C05487=1208.103,115.471,-50.349,-178.483,5.857,148.589
C05488=1208.098,115.720,-50.368,-178.480,5.858,148.588
C05489=1208.094,115.969,-50.387,-178.477,5.859,148.588
C05490=1208.089,116.219,-50.407,-178.474,5.860,148.587
C05491=1208.084,116.468,-50.426,-178.472,5.861,148.587
C05492=1208.079,116.717,-50.447,-178.469,5.863,148.586
C05493=1208.074,116.965,-50.466,-178.467,5.864,148.586
C05494=1208.070,117.215,-50.485,-178.465,5.865,148.585
C05495=1208.065,117.464,-50.505,-178.461,5.866,148.585
C05496=1208.060,117.713,-50.524,-178.459,5.867,148.584
C05497=1208.055,117.963,-50.543,-178.456,5.868,148.584
C05498=1208.051,118.212,-50.563,-178.454,5.869,148.583
C05499=1208.046,118.461,-50.582,-178.451,5.871,148.583
C05500=1208.041,118.710,-50.602,-178.449,5.872,148.582
C05501=1208.036,118.960,-50.621,-178.446,5.872,148.582
C05502=1208.031,119.209,-50.640,-178.443,5.874,148.581
C05503=1208.026,119.458,-50.660,-178.441,5.875,148.581
C05504=1208.021,119.707,-50.680,-178.438,5.877,148.580
C05505=1208.017,119.956,-50.699,-178.436,5.877,148.580
C05506=1208.013,120.205,-50.719,-178.433,5.879,148.579
C05507=1208.007,120.454,-50.738,-178.431,5.880,148.579
C05508=1208.002,120.704,-50.758,-178.428,5.881,148.578
C05509=1207.998,120.953,-50.778,-178.425,5.882,148.578
C05510=1207.993,121.202,-50.798,-178.423,5.883,148.577
C05511=1207.988,121.451,-50.817,-178.420,5.885,148.577
C05512=1207.983,121.701,-50.837,-178.418,5.885,148.576
C05513=1207.979,121.950,-50.856,-178.415,5.887,148.576
C05514=1207.974,122.198,-50.876,-178.412,5.888,148.575
C05515=1207.969,122.448,-50.895,-178.410,5.889,148.575
C05516=1207.965,122.698,-50.915,-178.407,5.890,148.574
C05517=1207.959,122.946,-50.934,-178.404,5.892,148.574
C05518=1207.955,123.195,-50.955,-178.402,5.893,148.573
C05519=1207.950,123.445,-50.974,-178.399,5.894,148.573
C05520=1207.945,123.694,-50.994,-178.397,5.895,148.572
C05521=1207.940,123.943,-51.014,-178.394,5.897,148.572
C05522=1207.936,124.192,-51.034,-178.392,5.897,148.571
C05523=1207.931,124.442,-51.053,-178.388,5.899,148.571
C05524=1207.926,124.691,-51.074,-178.386,5.900,148.570
C05525=1207.921,124.940,-51.093,-178.384,5.901,148.570
C05526=1207.916,125.189,-51.113,-178.381,5.902,148.569
C05527=1207.912,125.438,-51.133,-178.379,5.903,148.569
C05528=1207.907,125.688,-51.153,-178.376,5.905,148.568
C05529=1207.902,125.937,-51.172,-178.374,5.906,148.568
C05530=1207.897,126.186,-51.192,-178.370,5.907,148.567
C05531=1207.893,126.435,-51.212,-178.368,5.908,148.567
C05532=1207.888,126.684,-51.232,-178.366,5.910,148.566
C05533=1207.883,126.933,-51.252,-178.363,5.910,148.566
C05534=1207.878,127.182,-51.272,-178.360,5.912,148.565
C05535=1207.874,127.431,-51.292,-178.358,5.913,148.565
C05536=1207.869,127.681,-51.311,-178.355,5.914,148.564
C05537=1207.864,127.930,-51.332,-178.353,5.915,148.564
C05538=1207.859,128.179,-51.351,-178.350,5.917,148.563
C05539=1207.855,128.428,-51.371,-178.348,5.918,148.563
C05540=1207.850,128.677,-51.391,-178.344,5.919,148.562
C05541=1207.846,128.926,-51.412,-178.342,5.920,148.562
C05542=1207.841,129.176,-51.431,-178.339,5.922,148.561
C05543=1207.836,129.425,-51.452,-178.337,5.923,148.561
C05544=1207.830,129.674,-51.471,-178.334,5.924,148.560
C05545=1207.826,129.923,-51.492,-178.332,5.925,148.560
C05546=1207.821,130.172,-51.512,-178.329,5.927,148.559
C05547=1207.817,130.421,-51.532,-178.326,5.927,148.559
C05548=1207.812,130.670,-51.552,-178.324,5.929,148.558
C05549=1207.807,130.920,-51.572,-178.322,5.930,148.558
C05550=1207.802,131.169,-51.592,-178.318,5.932,148.557
C05551=1207.797,131.418,-51.613,-178.316,5.933,148.557
C05552=1207.793,131.667,-51.632,-178.313,5.934,148.556
C05553=1207.788,131.916,-51.653,-178.311,5.935,148.556
C05554=1207.783,132.166,-51.672,-178.308,5.937,148.555
C05555=1207.779,132.415,-51.693,-178.306,5.937,148.555
C05556=1207.774,132.664,-51.714,-178.303,5.939,148.554
C05557=1207.769,132.932,-51.735,-178.300,5.941,148.554
C05558=1207.763,133.201,-51.757,-178.298,5.941,148.553
C05559=1207.759,133.469,-51.778,-178.295,5.943,148.553
C05560=1207.753,133.738,-51.801,-178.292,5.945,148.552
C05561=1207.748,133.987,-51.820,-178.289,5.945,148.552
C05562=1207.744,134.236,-51.841,-178.287,5.947,148.551
C05563=1207.739,134.486,-51.862,-178.285,5.948,148.551
C05564=1207.734,134.735,-51.881,-178.281,5.950,148.550
C05565=1207.730,134.984,-51.902,-178.279,5.951,148.550
C05566=1207.725,135.233,-51.922,-178.276,5.952,148.549
C05567=1207.719,135.482,-51.943,-178.273,5.954,148.549
C05568=1207.715,135.731,-51.962,-178.271,5.955,148.549
C05569=1207.710,135.980,-51.983,-178.268,5.956,148.548
C05570=1207.705,136.229,-52.004,-178.266,5.957,148.548
C05571=1207.701,136.478,-52.024,-178.263,5.959,148.547
C05572=1207.696,136.727,-52.045,-178.261,5.959,148.547
C05573=1207.691,136.977,-52.064,-178.258,5.961,148.546
C05574=1207.686,137.226,-52.085,-178.255,5.962,148.546
C05575=1207.682,137.475,-52.106,-178.253,5.964,148.545
C05576=1207.677,137.724,-52.126,-178.250,5.965,148.545
C05577=1207.672,137.973,-52.147,-178.247,5.966,148.544
C05578=1207.668,138.222,-52.167,-178.245,5.968,148.544
C05579=1207.663,138.471,-52.188,-178.243,5.969,148.543
C05580=1207.658,138.720,-52.209,-178.239,5.970,148.543
C05581=1207.653,138.970,-52.228,-178.237,5.971,148.542
C05582=1207.648,139.219,-52.249,-178.235,5.973,148.542
C05583=1207.644,139.468,-52.270,-178.232,5.974,148.541
C05584=1207.639,139.717,-52.290,-178.229,5.975,148.541
C05585=1207.634,139.966,-52.311,-178.227,5.977,148.541
C05586=1207.630,140.215,-52.331,-178.224,5.978,148.540
C05587=1207.625,140.464,-52.352,-178.221,5.980,148.540
C05588=1207.620,140.714,-52.373,-178.219,5.981,148.539
C05589=1207.616,140.962,-52.393,-178.216,5.982,148.539
C05590=1207.611,141.212,-52.414,-178.214,5.983,148.538
C05591=1207.606,141.461,-52.434,-178.211,5.985,148.538
C05592=1207.601,141.710,-52.455,-178.208,5.986,148.537
C05593=1207.597,141.959,-52.476,-178.206,5.987,148.537
C05594=1207.592,142.208,-52.496,-178.203,5.989,148.536
C05595=1207.587,142.457,-52.517,-178.201,5.990,148.536
C05596=1207.582,142.706,-52.537,-178.198,5.991,148.535
C05597=1207.577,142.955,-52.558,-178.195,5.993,148.535
C05598=1207.573,143.204,-52.579,-178.193,5.994,148.534
C05599=1207.568,143.454,-52.600,-178.190,5.996,148.534
C05600=1207.563,143.702,-52.620,-178.188,5.996,148.534
C05601=1207.559,143.952,-52.642,-178.185,5.998,148.533
C05602=1207.555,144.201,-52.662,-178.182,6.000,148.533
C05603=1207.549,144.450,-52.683,-178.180,6.001,148.532
C05604=1207.545,144.699,-52.704,-178.177,6.002,148.532
C05605=1207.540,144.948,-52.725,-178.175,6.003,148.531
C05606=1207.535,145.197,-52.745,-178.172,6.005,148.531
C05607=1207.530,145.446,-52.766,-178.169,6.006,148.530
C05608=1207.526,145.695,-52.787,-178.167,6.007,148.530
C05609=1207.521,145.944,-52.808,-178.164,6.009,148.529
C05610=1207.516,146.193,-52.829,-178.162,6.010,148.529
C05611=1207.512,146.443,-52.850,-178.159,6.012,148.528
C05612=1207.507,146.692,-52.871,-178.156,6.013,148.528
C05613=1207.503,146.941,-52.892,-178.154,6.014,148.528
C05614=1207.497,147.190,-52.913,-178.151,6.016,148.527
C05615=1207.493,147.439,-52.933,-178.149,6.017,148.527
C05616=1207.488,147.688,-52.954,-178.146,6.018,148.526
C05617=1207.483,147.937,-52.976,-178.143,6.020,148.526
C05618=1207.478,148.186,-52.996,-178.141,6.021,148.525
C05619=1207.474,148.436,-53.018,-178.138,6.023,148.525
C05620=1207.469,148.685,-53.039,-178.136,6.024,148.525
C05621=1207.465,148.933,-53.060,-178.133,6.025,148.524
C05622=1207.459,149.182,-53.081,-178.130,6.027,148.524
C05623=1207.455,149.431,-53.101,-178.128,6.028,148.523
C05624=1207.450,149.680,-53.123,-178.125,6.029,148.523
C05625=1207.446,149.930,-53.144,-178.122,6.031,148.522
C05626=1207.441,150.179,-53.164,-178.120,6.032,148.522
C05627=1207.436,150.428,-53.186,-178.118,6.034,148.521
C05628=1207.431,150.677,-53.207,-178.114,6.035,148.521
C05629=1207.427,150.925,-53.228,-178.112,6.036,148.520
C05630=1207.422,151.175,-53.249,-178.110,6.038,148.520
C05631=1207.417,151.424,-53.270,-178.107,6.039,148.519
C05632=1207.412,151.673,-53.292,-178.104,6.041,148.519
C05633=1207.408,151.922,-53.313,-178.102,6.042,148.519
C05634=1207.403,152.171,-53.334,-178.100,6.043,148.518
C05635=1207.398,152.421,-53.356,-178.096,6.045,148.518
C05636=1207.394,152.669,-53.377,-178.094,6.047,148.517
C05637=1207.389,152.918,-53.398,-178.092,6.047,148.517
C05638=1207.384,153.167,-53.419,-178.089,6.049,148.517
C05639=1207.380,153.417,-53.441,-178.086,6.051,148.516
C05640=1207.374,153.666,-53.462,-178.084,6.052,148.516
C05641=1207.370,153.914,-53.483,-178.081,6.054,148.515
C05642=1207.365,154.163,-53.504,-178.078,6.055,148.515
C05643=1207.361,154.413,-53.526,-178.076,6.056,148.514
C05644=1207.356,154.662,-53.547,-178.073,6.058,148.514
C05645=1207.351,154.911,-53.568,-178.070,6.060,148.513
C05646=1207.347,155.159,-53.589,-178.068,6.061,148.513
C05647=1207.342,155.409,-53.611,-178.065,6.062,148.512
C05648=1207.337,155.658,-53.632,-178.063,6.064,148.512
C05649=1207.332,155.907,-53.653,-178.060,6.065,148.512
C05650=1207.327,156.156,-53.675,-178.058,6.067,148.511
C05651=1207.323,156.405,-53.697,-178.055,6.068,148.511
C05652=1207.319,156.654,-53.717,-178.052,6.069,148.510
C05653=1207.314,156.903,-53.739,-178.050,6.071,148.510
C05654=1207.309,157.153,-53.760,-178.047,6.073,148.510
C05655=1207.304,157.401,-53.782,-178.045,6.073,148.509
C05656=1207.299,157.650,-53.804,-178.042,6.075,148.509
C05657=1207.295,157.900,-53.825,-178.039,6.077,148.508
C05658=1207.290,158.148,-53.847,-178.037,6.078,148.508
C05659=1207.285,158.397,-53.869,-178.034,6.079,148.507
C05660=1207.282,158.646,-53.890,-178.031,6.081,148.507
C05661=1207.276,158.915,-53.913,-178.029,6.083,148.506
C05662=1207.270,159.184,-53.936,-178.025,6.084,148.506
C05663=1207.265,159.453,-53.959,-178.023,6.086,148.505
C05664=1207.260,159.722,-53.983,-178.021,6.087,148.505
C05665=1207.256,159.971,-54.005,-178.018,6.089,148.505
C05666=1207.251,160.221,-54.026,-178.015,6.090,148.504
C05667=1207.247,160.470,-54.048,-178.012,6.092,148.504
C05668=1207.242,160.718,-54.069,-178.010,6.093,148.503
C05669=1207.237,160.967,-54.091,-178.007,6.095,148.503
C05670=1207.233,161.217,-54.112,-178.004,6.096,148.502
C05671=1207.228,161.465,-54.134,-178.002,6.097,148.502
C05672=1207.223,161.714,-54.156,-177.999,6.099,148.502
C05673=1207.219,161.963,-54.178,-177.997,6.101,148.501
C05674=1207.214,162.212,-54.199,-177.994,6.102,148.501
C05675=1207.210,162.461,-54.222,-177.992,6.103,148.500
C05676=1207.205,162.710,-54.243,-177.989,6.105,148.500
C05677=1207.200,162.959,-54.264,-177.986,6.107,148.500
C05678=1207.195,163.209,-54.286,-177.984,6.108,148.499
C05679=1207.190,163.457,-54.308,-177.981,6.109,148.499
C05680=1207.185,163.707,-54.331,-177.978,6.111,148.498
C05681=1207.181,163.956,-54.352,-177.976,6.113,148.498
C05682=1207.176,164.205,-54.374,-177.974,6.114,148.497
C05683=1207.171,164.454,-54.396,-177.971,6.116,148.497
C05684=1207.167,164.702,-54.418,-177.968,6.117,148.496
C05685=1207.162,164.952,-54.440,-177.966,6.118,148.496
C05686=1207.157,165.200,-54.461,-177.963,6.120,148.496
C05687=1207.153,165.450,-54.483,-177.960,6.122,148.495
C05688=1207.148,165.698,-54.505,-177.958,6.124,148.495
C05689=1207.144,165.947,-54.527,-177.955,6.124,148.494
C05690=1207.139,166.196,-54.549,-177.952,6.126,148.494
C05691=1207.135,166.445,-54.571,-177.950,6.128,148.494
C05692=1207.129,166.694,-54.593,-177.947,6.130,148.493
C05693=1207.125,166.944,-54.615,-177.945,6.131,148.493
C05694=1207.120,167.192,-54.637,-177.942,6.132,148.493
C05695=1207.116,167.442,-54.659,-177.939,6.134,148.492
C05696=1207.111,167.690,-54.681,-177.936,6.136,148.492
C05697=1207.107,167.940,-54.703,-177.934,6.137,148.491
C05698=1207.101,168.189,-54.725,-177.932,6.139,148.491
C05699=1207.097,168.438,-54.747,-177.929,6.140,148.490
C05700=1207.092,168.686,-54.769,-177.926,6.142,148.490
C05701=1207.088,168.935,-54.791,-177.924,6.143,148.489
C05702=1207.083,169.184,-54.813,-177.921,6.145,148.489
C05703=1207.078,169.434,-54.836,-177.918,6.146,148.489
C05704=1207.073,169.682,-54.857,-177.916,6.148,148.488
C05705=1207.069,169.932,-54.879,-177.914,6.149,148.488
C05706=1207.064,170.180,-54.901,-177.911,6.151,148.488
C05707=1207.060,170.429,-54.924,-177.908,6.152,148.487
C05708=1207.055,170.678,-54.946,-177.905,6.154,148.487
C05709=1207.050,170.927,-54.968,-177.903,6.155,148.486
C05710=1207.045,171.176,-54.990,-177.900,6.157,148.486
C05711=1207.041,171.425,-55.013,-177.898,6.159,148.486
C05712=1207.036,171.674,-55.035,-177.895,6.161,148.485
C05713=1207.032,171.923,-55.057,-177.892,6.162,148.485
C05714=1207.027,172.172,-55.079,-177.890,6.163,148.484
C05715=1207.022,172.421,-55.102,-177.887,6.165,148.484
C05716=1207.018,172.670,-55.124,-177.884,6.167,148.484
C05717=1207.013,172.919,-55.146,-177.882,6.169,148.483
C05718=1207.008,173.168,-55.168,-177.880,6.170,148.483
C05719=1207.003,173.416,-55.191,-177.877,6.171,148.482
C05720=1206.999,173.666,-55.213,-177.874,6.173,148.482
C05721=1206.994,173.915,-55.236,-177.871,6.175,148.481
C05722=1206.989,174.163,-55.258,-177.869,6.176,148.481
C05723=1206.985,174.413,-55.280,-177.866,6.177,148.481
C05724=1206.980,174.662,-55.303,-177.864,6.179,148.480
C05725=1206.976,174.910,-55.325,-177.861,6.181,148.480
C05726=1206.971,175.160,-55.347,-177.859,6.183,148.480
C05727=1206.966,175.408,-55.370,-177.856,6.185,148.479
C05728=1206.962,175.657,-55.392,-177.854,6.186,148.479
C05729=1206.957,175.907,-55.415,-177.851,6.187,148.478
C05730=1206.952,176.155,-55.437,-177.848,6.189,148.478
C05731=1206.948,176.404,-55.459,-177.845,6.191,148.478
C05732=1206.943,176.653,-55.483,-177.843,6.193,148.477
C05733=1206.938,176.902,-55.504,-177.841,6.193,148.477
C05734=1206.934,177.151,-55.528,-177.838,6.195,148.476
C05735=1206.929,177.400,-55.550,-177.835,6.197,148.476
C05736=1206.925,177.648,-55.572,-177.833,6.199,148.476
C05737=1206.920,177.898,-55.595,-177.830,6.201,148.475
C05738=1206.916,178.147,-55.617,-177.827,6.201,148.475
C05739=1206.910,178.396,-55.640,-177.825,6.203,148.474
C05740=1206.906,178.644,-55.662,-177.822,6.205,148.474
C05741=1206.901,178.894,-55.685,-177.819,6.207,148.474
C05742=1206.897,179.142,-55.708,-177.817,6.209,148.473
C05743=1206.892,179.391,-55.731,-177.814,6.210,148.473
C05744=1206.888,179.640,-55.753,-177.812,6.211,148.473
C05745=1206.882,179.889,-55.776,-177.809,6.213,148.472
C05746=1206.878,180.138,-55.798,-177.807,6.215,148.472
C05747=1206.874,180.387,-55.821,-177.804,6.217,148.472
C05748=1206.870,180.636,-55.844,-177.801,6.219,148.471
C05749=1206.864,180.885,-55.866,-177.798,6.220,148.471
C05750=1206.860,181.134,-55.889,-177.796,6.221,148.470
C05751=1206.855,181.383,-55.912,-177.793,6.223,148.470
C05752=1206.851,181.632,-55.935,-177.791,6.225,148.470
C05753=1206.846,181.880,-55.958,-177.788,6.227,148.469
C05754=1206.841,182.129,-55.981,-177.785,6.228,148.469
C05755=1206.837,182.379,-56.003,-177.783,6.230,148.468
C05756=1206.832,182.628,-56.026,-177.781,6.231,148.468
C05757=1206.827,182.876,-56.049,-177.778,6.233,148.468
C05758=1206.822,183.125,-56.071,-177.775,6.235,148.467
C05759=1206.818,183.374,-56.095,-177.773,6.237,148.467
C05760=1206.814,183.623,-56.117,-177.770,6.238,148.467
C05761=1206.809,183.871,-56.140,-177.767,6.240,148.466
C05762=1206.804,184.121,-56.163,-177.764,6.242,148.466
C05763=1206.800,184.370,-56.186,-177.762,6.243,148.465
C05764=1206.795,184.619,-56.209,-177.759,6.245,148.465
C05765=1206.790,184.888,-56.234,-177.757,6.246,148.465
C05766=1206.785,185.158,-56.259,-177.754,6.248,148.464
C05767=1206.780,185.428,-56.284,-177.751,6.251,148.464
C05768=1206.775,185.697,-56.308,-177.748,6.252,148.463
C05769=1206.770,185.946,-56.332,-177.745,6.254,148.463
C05770=1206.766,186.195,-56.355,-177.743,6.255,148.463
C05771=1206.761,186.443,-56.377,-177.740,6.257,148.462
C05772=1206.756,186.692,-56.401,-177.738,6.259,148.462
C05773=1206.752,186.941,-56.424,-177.735,6.261,148.462
C05774=1206.748,187.190,-56.447,-177.732,6.262,148.461
C05775=1206.743,187.439,-56.470,-177.730,6.264,148.461
C05776=1206.738,187.689,-56.493,-177.727,6.266,148.461
C05777=1206.733,187.937,-56.516,-177.724,6.268,148.460
C05778=1206.729,188.186,-56.539,-177.722,6.269,148.460
C05779=1206.724,188.435,-56.562,-177.720,6.271,148.459
C05780=1206.719,188.684,-56.585,-177.717,6.272,148.459
C05781=1206.715,188.933,-56.609,-177.714,6.274,148.459
C05782=1206.711,189.182,-56.631,-177.712,6.276,148.458
C05783=1206.706,189.431,-56.655,-177.709,6.278,148.458
C05784=1206.701,189.680,-56.678,-177.706,6.280,148.458
C05785=1206.696,189.928,-56.701,-177.704,6.282,148.457
C05786=1206.691,190.177,-56.724,-177.701,6.283,148.457
C05787=1206.687,190.426,-56.747,-177.699,6.284,148.457
C05788=1206.683,190.675,-56.771,-177.696,6.286,148.456
C05789=1206.678,190.924,-56.794,-177.694,6.288,148.456
C05790=1206.674,191.172,-56.818,-177.691,6.290,148.456
C05791=1206.669,191.421,-56.841,-177.688,6.292,148.455
C05792=1206.664,191.670,-56.865,-177.686,6.293,148.455
C05793=1206.660,191.919,-56.887,-177.683,6.295,148.455
C05794=1206.655,192.168,-56.911,-177.680,6.297,148.454
C05795=1206.651,192.417,-56.934,-177.678,6.299,148.454
C05796=1206.645,192.666,-56.957,-177.675,6.301,148.454
C05797=1206.641,192.915,-56.981,-177.672,6.303,148.453
C05798=1206.636,193.163,-57.005,-177.670,6.304,148.453
C05799=1206.632,193.412,-57.028,-177.668,6.305,148.452
C05800=1206.627,193.661,-57.051,-177.665,6.307,148.452
C05801=1206.622,193.910,-57.075,-177.662,6.309,148.452
C05802=1206.618,194.159,-57.097,-177.660,6.311,148.451
C05803=1206.614,194.408,-57.121,-177.657,6.313,148.451
C05804=1206.609,194.656,-57.145,-177.654,6.314,148.451
C05805=1206.605,194.905,-57.168,-177.652,6.316,148.450
C05806=1206.600,195.154,-57.192,-177.649,6.318,148.450
C05807=1206.595,195.403,-57.215,-177.647,6.320,148.450
C05808=1206.591,195.652,-57.239,-177.644,6.322,148.449
C05809=1206.586,195.901,-57.262,-177.641,6.324,148.449
C05810=1206.581,196.150,-57.286,-177.639,6.325,148.449
C05811=1206.577,196.398,-57.310,-177.636,6.326,148.448
C05812=1206.572,196.647,-57.333,-177.634,6.328,148.448
C05813=1206.568,196.896,-57.357,-177.631,6.330,148.448
C05814=1206.563,197.145,-57.381,-177.629,6.332,148.447
C05815=1206.558,197.394,-57.404,-177.626,6.334,148.447
C05816=1206.554,197.643,-57.427,-177.623,6.336,148.447
C05817=1206.549,197.891,-57.451,-177.621,6.337,148.446
C05818=1206.545,198.140,-57.475,-177.618,6.339,148.446
C05819=1206.540,198.389,-57.498,-177.615,6.341,148.445
C05820=1206.536,198.638,-57.522,-177.613,6.343,148.445
C05821=1206.531,198.887,-57.546,-177.610,6.345,148.445
C05822=1206.526,199.135,-57.570,-177.607,6.346,148.444
C05823=1206.522,199.385,-57.594,-177.605,6.348,148.444
C05824=1206.517,199.634,-57.618,-177.602,6.350,148.444
C05825=1206.513,199.883,-57.641,-177.599,6.352,148.443
C05826=1206.508,200.131,-57.665,-177.597,6.354,148.443
C05827=1206.503,200.380,-57.689,-177.594,6.356,148.443
C05828=1206.499,200.629,-57.712,-177.591,6.357,148.442
C05829=1206.494,200.877,-57.736,-177.589,6.359,148.442
C05830=1206.490,201.126,-57.760,-177.586,6.361,148.442
C05831=1206.485,201.375,-57.784,-177.583,6.363,148.441
C05832=1206.481,201.623,-57.808,-177.581,6.365,148.441
C05833=1206.475,201.873,-57.832,-177.578,6.367,148.441
C05834=1206.472,202.122,-57.856,-177.576,6.368,148.440
C05835=1206.467,202.371,-57.880,-177.573,6.371,148.440
C05836=1206.463,202.619,-57.904,-177.571,6.372,148.440
C05837=1206.458,202.868,-57.927,-177.569,6.373,148.439
C05838=1206.453,203.117,-57.951,-177.566,6.375,148.439
C05839=1206.448,203.365,-57.976,-177.563,6.377,148.439
C05840=1206.444,203.614,-57.999,-177.561,6.379,148.438
C05841=1206.439,203.863,-58.023,-177.558,6.381,148.438
C05842=1206.435,204.112,-58.048,-177.555,6.383,148.438
C05843=1206.431,204.361,-58.071,-177.553,6.384,148.437
C05844=1206.426,204.610,-58.096,-177.550,6.386,148.437
C05845=1206.421,204.858,-58.120,-177.547,6.388,148.437
C05846=1206.416,205.107,-58.143,-177.545,6.390,148.436
C05847=1206.412,205.356,-58.167,-177.542,6.392,148.436
C05848=1206.408,205.605,-58.192,-177.539,6.393,148.436
C05849=1206.403,205.854,-58.216,-177.537,6.395,148.435
C05850=1206.398,206.102,-58.240,-177.535,6.397,148.435
C05851=1206.393,206.351,-58.264,-177.532,6.399,148.435
C05852=1206.389,206.600,-58.288,-177.529,6.401,148.435
C05853=1206.385,206.849,-58.312,-177.527,6.403,148.434
C05854=1206.380,207.098,-58.336,-177.524,6.405,148.434
C05855=1206.375,207.346,-58.361,-177.521,6.407,148.434
C05856=1206.371,207.595,-58.385,-177.519,6.408,148.433
C05857=1206.367,207.843,-58.409,-177.516,6.410,148.433
C05858=1206.362,208.093,-58.433,-177.513,6.413,148.433
C05859=1206.357,208.342,-58.457,-177.510,6.415,148.432
C05860=1206.353,208.590,-58.481,-177.508,6.417,148.432
C05861=1206.348,208.839,-58.506,-177.506,6.419,148.432
C05862=1206.344,209.088,-58.531,-177.503,6.421,148.431
C05863=1206.339,209.337,-58.555,-177.500,6.422,148.431
C05864=1206.334,209.586,-58.579,-177.498,6.424,148.431
C05865=1206.330,209.834,-58.603,-177.495,6.426,148.430
C05866=1206.325,210.084,-58.628,-177.492,6.428,148.430
C05867=1206.321,210.332,-58.652,-177.490,6.430,148.430
C05868=1206.316,210.580,-58.676,-177.487,6.432,148.429
C05869=1206.311,210.851,-58.703,-177.484,6.433,148.429
C05870=1206.306,211.121,-58.729,-177.482,6.435,148.429
C05871=1206.301,211.392,-58.756,-177.478,6.438,148.428
C05872=1206.296,211.662,-58.782,-177.476,6.440,148.428
C05873=1206.292,211.911,-58.806,-177.473,6.442,148.428
C05874=1206.287,212.160,-58.831,-177.471,6.443,148.427
C05875=1206.283,212.409,-58.856,-177.468,6.446,148.427
C05876=1206.278,212.657,-58.880,-177.466,6.447,148.427
C05877=1206.273,212.906,-58.904,-177.463,6.449,148.427
C05878=1206.269,213.155,-58.929,-177.460,6.451,148.426
C05879=1206.264,213.404,-58.953,-177.458,6.453,148.426
C05880=1206.260,213.652,-58.979,-177.455,6.455,148.426
C05881=1206.256,213.901,-59.003,-177.453,6.457,148.425
C05882=1206.251,214.150,-59.028,-177.450,6.458,148.425
C05883=1206.246,214.398,-59.052,-177.447,6.461,148.425
C05884=1206.242,214.647,-59.077,-177.445,6.463,148.425
C05885=1206.237,214.896,-59.101,-177.442,6.465,148.424
C05886=1206.232,215.145,-59.126,-177.439,6.467,148.424
C05887=1206.228,215.394,-59.150,-177.437,6.469,148.424
C05888=1206.223,215.642,-59.175,-177.434,6.471,148.423
C05889=1206.220,215.891,-59.200,-177.431,6.472,148.423
C05890=1206.215,216.140,-59.225,-177.429,6.475,148.423
C05891=1206.209,216.388,-59.249,-177.427,6.476,148.422
C05892=1206.206,216.637,-59.274,-177.424,6.478,148.422
C05893=1206.201,216.886,-59.298,-177.421,6.480,148.422
C05894=1206.196,217.134,-59.323,-177.419,6.482,148.421
C05895=1206.192,217.383,-59.348,-177.416,6.484,148.421
C05896=1206.187,217.632,-59.373,-177.414,6.486,148.421
C05897=1206.183,217.881,-59.397,-177.411,6.489,148.421
C05898=1206.178,218.129,-59.423,-177.408,6.490,148.420
C05899=1206.174,218.378,-59.447,-177.405,6.492,148.420
C05900=1206.169,218.627,-59.472,-177.403,6.494,148.420
C05901=1206.164,218.875,-59.497,-177.400,6.496,148.419
C05902=1206.161,219.124,-59.522,-177.398,6.498,148.419
C05903=1206.156,219.373,-59.546,-177.395,6.500,148.419
C05904=1206.151,219.622,-59.572,-177.393,6.502,148.419
C05905=1206.147,219.870,-59.596,-177.390,6.504,148.418
C05906=1206.142,220.120,-59.621,-177.387,6.505,148.418
C05907=1206.138,220.368,-59.647,-177.385,6.507,148.418
C05908=1206.133,220.616,-59.671,-177.383,6.509,148.418
C05909=1206.129,220.866,-59.696,-177.379,6.512,148.417
C05910=1206.124,221.114,-59.721,-177.377,6.514,148.417
C05911=1206.119,221.363,-59.746,-177.374,6.516,148.417
C05912=1206.115,221.611,-59.771,-177.371,6.518,148.416
C05913=1206.111,221.860,-59.796,-177.369,6.520,148.416
C05914=1206.106,222.109,-59.821,-177.367,6.522,148.416
C05915=1206.101,222.358,-59.846,-177.364,6.523,148.415
C05916=1206.097,222.606,-59.871,-177.361,6.525,148.415
C05917=1206.093,222.855,-59.896,-177.359,6.527,148.415
C05918=1206.088,223.103,-59.922,-177.357,6.529,148.415
C05919=1206.083,223.353,-59.947,-177.353,6.532,148.414
C05920=1206.078,223.601,-59.972,-177.351,6.534,148.414
C05921=1206.075,223.850,-59.996,-177.348,6.536,148.414
C05922=1206.070,224.098,-60.022,-177.345,6.537,148.413
C05923=1206.065,224.347,-60.047,-177.343,6.540,148.413
C05924=1206.060,224.596,-60.072,-177.341,6.541,148.413
C05925=1206.056,224.845,-60.097,-177.338,6.543,148.413
C05926=1206.052,225.093,-60.122,-177.335,6.545,148.412
C05927=1206.048,225.342,-60.148,-177.333,6.547,148.412
C05928=1206.043,225.591,-60.173,-177.330,6.550,148.412
C05929=1206.038,225.839,-60.198,-177.327,6.552,148.412
C05930=1206.034,226.089,-60.223,-177.325,6.554,148.411
C05931=1206.029,226.337,-60.249,-177.323,6.556,148.411
C05932=1206.025,226.585,-60.274,-177.320,6.558,148.411
C05933=1206.020,226.834,-60.299,-177.317,6.560,148.411
C05934=1206.016,227.083,-60.324,-177.315,6.561,148.410
C05935=1206.012,227.331,-60.350,-177.313,6.564,148.410
C05936=1206.007,227.580,-60.375,-177.310,6.565,148.410
C05937=1206.003,227.829,-60.400,-177.307,6.568,148.410
C05938=1205.998,228.077,-60.426,-177.304,6.570,148.409
C05939=1205.993,228.326,-60.452,-177.302,6.572,148.409
C05940=1205.988,228.575,-60.476,-177.299,6.574,148.409
C05941=1205.984,228.823,-60.502,-177.297,6.576,148.408
C05942=1205.980,229.072,-60.528,-177.294,6.578,148.408
C05943=1205.975,229.320,-60.553,-177.292,6.580,148.408
C05944=1205.971,229.570,-60.578,-177.289,6.582,148.408
C05945=1205.966,229.819,-60.604,-177.286,6.584,148.407
C05946=1205.961,230.067,-60.629,-177.283,6.586,148.407
C05947=1205.957,230.315,-60.655,-177.281,6.588,148.407
C05948=1205.952,230.564,-60.680,-177.279,6.590,148.407
C05949=1205.948,230.812,-60.706,-177.276,6.592,148.406
C05950=1205.944,231.062,-60.731,-177.273,6.594,148.406
C05951=1205.939,231.310,-60.757,-177.271,6.596,148.406
C05952=1205.935,231.559,-60.782,-177.268,6.599,148.406
C05953=1205.930,231.808,-60.808,-177.265,6.600,148.405
C05954=1205.926,232.056,-60.833,-177.263,6.603,148.405
C05955=1205.921,232.304,-60.859,-177.261,6.604,148.405
C05956=1205.917,232.553,-60.885,-177.258,6.606,148.405
C05957=1205.912,232.801,-60.910,-177.256,6.609,148.404
C05958=1205.908,233.050,-60.936,-177.253,6.611,148.404
C05959=1205.904,233.299,-60.962,-177.250,6.613,148.404
C05960=1205.899,233.548,-60.988,-177.247,6.615,148.403
C05961=1205.894,233.796,-61.014,-177.245,6.617,148.403
C05962=1205.890,234.045,-61.039,-177.243,6.619,148.403
C05963=1205.886,234.294,-61.065,-177.240,6.621,148.403
C05964=1205.881,234.542,-61.090,-177.237,6.624,148.403
C05965=1205.877,234.791,-61.116,-177.235,6.626,148.402
C05966=1205.872,235.039,-61.142,-177.232,6.627,148.402
C05967=1205.868,235.288,-61.167,-177.230,6.630,148.402
C05968=1205.863,235.537,-61.194,-177.227,6.631,148.402
C05969=1205.858,235.786,-61.219,-177.224,6.633,148.401
C05970=1205.854,236.034,-61.245,-177.222,6.636,148.401
C05971=1205.849,236.282,-61.271,-177.219,6.638,148.401
C05972=1205.845,236.531,-61.296,-177.217,6.640,148.401
C05973=1205.841,236.802,-61.325,-177.214,6.642,148.400
C05974=1205.835,237.074,-61.353,-177.211,6.645,148.400
C05975=1205.830,237.346,-61.381,-177.209,6.647,148.400
C05976=1205.826,237.617,-61.410,-177.205,6.649,148.400
C05977=1205.821,237.866,-61.436,-177.203,6.651,148.399
C05978=1205.816,238.114,-61.461,-177.201,6.653,148.399
C05979=1205.812,238.363,-61.488,-177.198,6.655,148.399
C05980=1205.808,238.611,-61.514,-177.195,6.657,148.399
C05981=1205.803,238.860,-61.540,-177.193,6.660,148.399
C05982=1205.799,239.109,-61.566,-177.190,6.662,148.398
C05983=1205.794,239.357,-61.592,-177.187,6.664,148.398
C05984=1205.789,239.606,-61.617,-177.185,6.666,148.398
C05985=1205.785,239.854,-61.644,-177.183,6.668,148.397
C05986=1205.780,240.104,-61.670,-177.179,6.670,148.397
C05987=1205.776,240.352,-61.696,-177.177,6.673,148.397
C05988=1205.772,240.600,-61.722,-177.175,6.674,148.397
C05989=1205.767,240.849,-61.748,-177.172,6.676,148.396
C05990=1205.763,241.098,-61.774,-177.170,6.679,148.396
C05991=1205.759,241.346,-61.801,-177.167,6.681,148.396
C05992=1205.754,241.595,-61.827,-177.164,6.683,148.396
C05993=1205.749,241.844,-61.853,-177.162,6.685,148.396
C05994=1205.745,242.091,-61.879,-177.159,6.687,148.395
C05995=1205.740,242.340,-61.905,-177.157,6.689,148.395
C05996=1205.736,242.589,-61.931,-177.154,6.692,148.395
C05997=1205.732,242.837,-61.957,-177.151,6.694,148.395
C05998=1205.727,243.087,-61.984,-177.149,6.696,148.395
C05999=1205.723,243.335,-62.010,-177.146,6.698,148.394
C06000=1205.718,243.584,-62.036,-177.144,6.701,148.394
C06001=1205.714,243.833,-62.062,-177.141,6.703,148.394
C06002=1205.709,244.080,-62.088,-177.138,6.705,148.394
C06003=1205.704,244.329,-62.115,-177.136,6.707,148.393
C06004=1205.700,244.577,-62.141,-177.134,6.709,148.393
C06005=1205.695,244.827,-62.167,-177.131,6.712,148.393
C06006=1205.691,245.075,-62.194,-177.128,6.713,148.393
C06007=1205.687,245.324,-62.220,-177.126,6.715,148.392
C06008=1205.683,245.572,-62.247,-177.124,6.717,148.392
C06009=1205.678,245.821,-62.273,-177.120,6.720,148.392
C06010=1205.674,246.069,-62.300,-177.118,6.722,148.392
C06011=1205.670,246.318,-62.326,-177.116,6.724,148.392
C06012=1205.665,246.567,-62.352,-177.113,6.726,148.391
C06013=1205.661,246.815,-62.379,-177.110,6.729,148.391
C06014=1205.656,247.064,-62.405,-177.108,6.731,148.391
C06015=1205.652,247.312,-62.432,-177.106,6.733,148.391
C06016=1205.647,247.560,-62.458,-177.103,6.735,148.391
C06017=1205.642,247.809,-62.485,-177.100,6.738,148.391
C06018=1205.638,248.057,-62.511,-177.098,6.740,148.390
C06019=1205.633,248.306,-62.538,-177.095,6.742,148.390
C06020=1205.629,248.555,-62.564,-177.093,6.744,148.390
C06021=1205.624,248.803,-62.591,-177.090,6.746,148.390
C06022=1205.620,249.051,-62.618,-177.087,6.749,148.389
C06023=1205.615,249.300,-62.644,-177.085,6.750,148.389
C06024=1205.611,249.549,-62.671,-177.083,6.753,148.389
C06025=1205.607,249.797,-62.697,-177.080,6.755,148.389
C06026=1205.602,250.046,-62.724,-177.077,6.757,148.388
C06027=1205.598,250.294,-62.750,-177.075,6.759,148.388
C06028=1205.593,250.543,-62.777,-177.072,6.761,148.388
C06029=1205.589,250.791,-62.804,-177.069,6.764,148.388
C06030=1205.585,251.039,-62.831,-177.067,6.766,148.388
C06031=1205.580,251.289,-62.857,-177.065,6.768,148.388
C06032=1205.575,251.537,-62.884,-177.062,6.770,148.387
C06033=1205.571,251.785,-62.911,-177.059,6.773,148.387
C06034=1205.567,252.034,-62.938,-177.057,6.775,148.387
C06035=1205.563,252.283,-62.965,-177.055,6.777,148.387
C06036=1205.558,252.532,-62.991,-177.051,6.780,148.387
C06037=1205.554,252.780,-63.018,-177.049,6.782,148.386
C06038=1205.549,253.029,-63.045,-177.047,6.784,148.386
C06039=1205.545,253.277,-63.072,-177.044,6.786,148.386
C06040=1205.540,253.525,-63.099,-177.041,6.789,148.386
C06041=1205.536,253.774,-63.126,-177.039,6.791,148.386
C06042=1205.532,254.022,-63.152,-177.036,6.793,148.385
C06043=1205.527,254.271,-63.179,-177.033,6.795,148.385
C06044=1205.523,254.519,-63.206,-177.031,6.798,148.385
C06045=1205.518,254.768,-63.233,-177.029,6.799,148.385
C06046=1205.514,255.016,-63.260,-177.026,6.802,148.385
C06047=1205.509,255.264,-63.287,-177.023,6.804,148.384
C06048=1205.505,255.513,-63.314,-177.021,6.807,148.384
C06049=1205.501,255.762,-63.341,-177.018,6.808,148.384
C06050=1205.497,256.010,-63.368,-177.016,6.811,148.384
C06051=1205.492,256.259,-63.395,-177.013,6.813,148.384
C06052=1205.487,256.507,-63.422,-177.011,6.815,148.384
C06053=1205.483,256.756,-63.449,-177.008,6.818,148.383
C06054=1205.478,257.004,-63.476,-177.006,6.820,148.383
C06055=1205.473,257.253,-63.503,-177.003,6.822,148.383
C06056=1205.470,257.502,-63.530,-177.000,6.825,148.383
C06057=1205.465,257.750,-63.557,-176.998,6.827,148.383
C06058=1205.461,257.999,-63.584,-176.996,6.829,148.382
C06059=1205.456,258.247,-63.611,-176.993,6.831,148.382
C06060=1205.451,258.495,-63.638,-176.990,6.834,148.382
C06061=1205.447,258.743,-63.666,-176.988,6.836,148.382
C06062=1205.443,258.993,-63.693,-176.985,6.838,148.382
C06063=1205.439,259.241,-63.720,-176.982,6.841,148.381
C06064=1205.434,259.489,-63.747,-176.980,6.843,148.381
C06065=1205.430,259.738,-63.774,-176.978,6.845,148.381
C06066=1205.425,259.986,-63.802,-176.975,6.848,148.381
C06067=1205.421,260.235,-63.829,-176.973,6.850,148.381
C06068=1205.417,260.483,-63.856,-176.970,6.852,148.381
C06069=1205.412,260.732,-63.883,-176.967,6.855,148.381
C06070=1205.407,260.980,-63.910,-176.965,6.857,148.380
C06071=1205.403,261.228,-63.938,-176.963,6.859,148.380
C06072=1205.399,261.477,-63.966,-176.959,6.862,148.380
C06073=1205.394,261.726,-63.993,-176.957,6.864,148.380
C06074=1205.390,261.974,-64.020,-176.955,6.866,148.380
C06075=1205.385,262.222,-64.047,-176.952,6.869,148.380
C06076=1205.381,262.471,-64.075,-176.950,6.871,148.379
C06077=1205.377,262.744,-64.105,-176.947,6.874,148.379
C06078=1205.372,263.016,-64.135,-176.943,6.876,148.379
C06079=1205.367,263.289,-64.165,-176.941,6.878,148.379
C06080=1205.362,263.562,-64.195,-176.938,6.881,148.379
C06081=1205.358,263.811,-64.222,-176.936,6.883,148.378
C06082=1205.353,264.058,-64.250,-176.933,6.886,148.378
C06083=1205.349,264.307,-64.277,-176.931,6.888,148.378
C06084=1205.345,264.556,-64.305,-176.928,6.890,148.378
C06085=1205.340,264.804,-64.332,-176.925,6.893,148.378
C06086=1205.336,265.052,-64.359,-176.923,6.895,148.378
C06087=1205.332,265.301,-64.388,-176.921,6.897,148.377
C06088=1205.326,265.550,-64.415,-176.918,6.900,148.377
C06089=1205.322,265.798,-64.443,-176.915,6.902,148.377
C06090=1205.317,266.046,-64.470,-176.913,6.905,148.377
C06091=1205.314,266.295,-64.498,-176.910,6.907,148.377
C06092=1205.309,266.543,-64.525,-176.908,6.909,148.377
C06093=1205.305,266.791,-64.553,-176.905,6.912,148.377
C06094=1205.301,267.040,-64.580,-176.903,6.914,148.376
C06095=1205.296,267.288,-64.608,-176.900,6.916,148.376
C06096=1205.291,267.537,-64.636,-176.898,6.919,148.376
C06097=1205.287,267.786,-64.664,-176.895,6.921,148.376
C06098=1205.283,268.033,-64.692,-176.892,6.924,148.376
C06099=1205.278,268.282,-64.719,-176.890,6.926,148.376
C06100=1205.274,268.531,-64.747,-176.888,6.928,148.375
C06101=1205.270,268.779,-64.774,-176.885,6.931,148.375
C06102=1205.265,269.027,-64.802,-176.882,6.933,148.375
C06103=1205.261,269.276,-64.831,-176.880,6.936,148.375
C06104=1205.256,269.524,-64.858,-176.877,6.938,148.375
C06105=1205.252,269.773,-64.886,-176.875,6.940,148.375
C06106=1205.248,270.021,-64.914,-176.872,6.943,148.375
C06107=1205.243,270.270,-64.941,-176.870,6.945,148.374
C06108=1205.239,270.518,-64.969,-176.867,6.948,148.374
C06109=1205.235,270.766,-64.997,-176.865,6.950,148.374
C06110=1205.231,271.015,-65.025,-176.862,6.952,148.374
C06111=1205.225,271.263,-65.053,-176.859,6.955,148.374
C06112=1205.221,271.511,-65.081,-176.857,6.957,148.374
C06113=1205.217,271.760,-65.109,-176.854,6.960,148.374
C06114=1205.212,272.008,-65.137,-176.852,6.962,148.374
C06115=1205.208,272.257,-65.165,-176.850,6.964,148.373
C06116=1205.204,272.505,-65.192,-176.847,6.967,148.373
C06117=1205.200,272.753,-65.220,-176.844,6.969,148.373
C06118=1205.195,273.002,-65.249,-176.842,6.972,148.373
C06119=1205.191,273.250,-65.277,-176.839,6.974,148.373
C06120=1205.187,273.498,-65.305,-176.836,6.977,148.373
C06121=1205.182,273.747,-65.333,-176.834,6.979,148.373
C06122=1205.178,273.996,-65.361,-176.832,6.981,148.372
C06123=1205.173,274.244,-65.388,-176.829,6.984,148.372
C06124=1205.169,274.492,-65.417,-176.827,6.986,148.372
C06125=1205.165,274.740,-65.445,-176.824,6.989,148.372
C06126=1205.160,274.989,-65.474,-176.822,6.991,148.372
C06127=1205.156,275.237,-65.502,-176.819,6.994,148.372
C06128=1205.152,275.486,-65.530,-176.816,6.996,148.372
C06129=1205.147,275.734,-65.558,-176.814,6.998,148.372
C06130=1205.143,275.982,-65.586,-176.811,7.001,148.371
C06131=1205.138,276.231,-65.615,-176.809,7.003,148.371
C06132=1205.134,276.479,-65.643,-176.806,7.006,148.371
C06133=1205.130,276.727,-65.670,-176.804,7.008,148.371
C06134=1205.126,276.976,-65.699,-176.801,7.011,148.371
C06135=1205.121,277.224,-65.727,-176.799,7.013,148.371
C06136=1205.117,277.473,-65.756,-176.796,7.016,148.371
C06137=1205.112,277.721,-65.783,-176.794,7.018,148.371
C06138=1205.108,277.969,-65.812,-176.791,7.020,148.370
C06139=1205.103,278.217,-65.840,-176.788,7.023,148.370
C06140=1205.099,278.466,-65.869,-176.786,7.025,148.370
C06141=1205.095,278.714,-65.897,-176.783,7.028,148.370
C06142=1205.090,278.963,-65.925,-176.781,7.030,148.370
C06143=1205.087,279.211,-65.954,-176.778,7.033,148.370
C06144=1205.082,279.459,-65.982,-176.776,7.036,148.370
C06145=1205.078,279.708,-66.011,-176.773,7.038,148.370
C06146=1205.073,279.956,-66.039,-176.771,7.040,148.370
C06147=1205.069,280.205,-66.067,-176.768,7.043,148.369
C06148=1205.064,280.453,-66.096,-176.766,7.046,148.369
C06149=1205.061,280.701,-66.124,-176.763,7.048,148.369
C06150=1205.056,280.950,-66.153,-176.761,7.050,148.369
C06151=1205.051,281.198,-66.181,-176.758,7.054,148.369
C06152=1205.047,281.446,-66.210,-176.756,7.056,148.369
C06153=1205.042,281.694,-66.239,-176.753,7.058,148.369
C06154=1205.039,281.942,-66.267,-176.751,7.061,148.369
C06155=1205.034,282.191,-66.296,-176.749,7.063,148.369
C06156=1205.029,282.440,-66.324,-176.746,7.066,148.369
C06157=1205.026,282.687,-66.353,-176.743,7.068,148.368
C06158=1205.021,282.936,-66.381,-176.741,7.071,148.368
C06159=1205.016,283.185,-66.410,-176.738,7.073,148.368
C06160=1205.013,283.432,-66.439,-176.736,7.076,148.368
C06161=1205.008,283.681,-66.467,-176.733,7.078,148.368
C06162=1205.003,283.930,-66.496,-176.730,7.081,148.368
C06163=1205.000,284.178,-66.525,-176.728,7.083,148.368
C06164=1204.995,284.426,-66.553,-176.726,7.086,148.368
C06165=1204.990,284.675,-66.582,-176.723,7.088,148.368
C06166=1204.987,284.923,-66.611,-176.720,7.091,148.367
C06167=1204.981,285.171,-66.639,-176.718,7.093,148.367
C06168=1204.977,285.419,-66.669,-176.715,7.096,148.367
C06169=1204.974,285.668,-66.697,-176.713,7.098,148.367
C06170=1204.969,285.915,-66.726,-176.710,7.101,148.367
C06171=1204.964,286.164,-66.755,-176.708,7.103,148.367
C06172=1204.960,286.412,-66.784,-176.705,7.106,148.367
C06173=1204.956,286.660,-66.812,-176.703,7.108,148.367
C06174=1204.952,286.908,-66.841,-176.700,7.111,148.367
C06175=1204.947,287.157,-66.870,-176.698,7.114,148.367
C06176=1204.943,287.406,-66.899,-176.695,7.116,148.366
C06177=1204.939,287.653,-66.927,-176.693,7.118,148.366
C06178=1204.934,287.902,-66.957,-176.690,7.122,148.366
C06179=1204.930,288.151,-66.985,-176.688,7.124,148.366
C06180=1204.925,288.398,-67.014,-176.686,7.127,148.366
C06181=1204.921,288.673,-67.046,-176.682,7.129,148.366
C06182=1204.916,288.948,-67.078,-176.680,7.132,148.366
C06183=1204.912,289.221,-67.110,-176.677,7.135,148.366
C06184=1204.906,289.496,-67.143,-176.674,7.138,148.366
C06185=1204.903,289.744,-67.172,-176.672,7.140,148.366
C06186=1204.898,289.993,-67.200,-176.669,7.143,148.366
C06187=1204.893,290.240,-67.229,-176.667,7.146,148.366
C06188=1204.889,290.489,-67.259,-176.664,7.149,148.366
C06189=1204.885,290.738,-67.288,-176.662,7.151,148.366
C06190=1204.880,290.986,-67.317,-176.659,7.154,148.366
C06191=1204.876,291.233,-67.346,-176.657,7.156,148.365
C06192=1204.872,291.482,-67.376,-176.654,7.159,148.365
C06193=1204.867,291.731,-67.404,-176.652,7.161,148.365
C06194=1204.864,291.979,-67.433,-176.649,7.164,148.365
C06195=1204.859,292.227,-67.463,-176.647,7.166,148.365
C06196=1204.855,292.474,-67.492,-176.644,7.169,148.365
C06197=1204.850,292.723,-67.520,-176.642,7.171,148.365
C06198=1204.846,292.972,-67.550,-176.640,7.174,148.365
C06199=1204.842,293.220,-67.579,-176.637,7.177,148.365
C06200=1204.838,293.468,-67.609,-176.634,7.179,148.365
C06201=1204.833,293.716,-67.638,-176.632,7.182,148.365
C06202=1204.829,293.964,-67.667,-176.629,7.184,148.365
C06203=1204.824,294.213,-67.696,-176.627,7.187,148.365
C06204=1204.820,294.461,-67.726,-176.625,7.190,148.364
C06205=1204.816,294.709,-67.755,-176.622,7.193,148.364
C06206=1204.812,294.958,-67.784,-176.620,7.195,148.364
C06207=1204.807,295.206,-67.814,-176.617,7.198,148.364
C06208=1204.803,295.454,-67.843,-176.615,7.200,148.364
C06209=1204.799,295.702,-67.873,-176.612,7.203,148.364
C06210=1204.794,295.950,-67.902,-176.610,7.206,148.364
C06211=1204.790,296.198,-67.931,-176.607,7.208,148.364
C06212=1204.786,296.446,-67.961,-176.604,7.211,148.364
C06213=1204.782,296.695,-67.990,-176.602,7.213,148.364
C06214=1204.778,296.943,-68.020,-176.599,7.216,148.364
C06215=1204.773,297.192,-68.050,-176.597,7.218,148.364
C06216=1204.768,297.440,-68.079,-176.595,7.221,148.364
C06217=1204.764,297.688,-68.109,-176.592,7.225,148.364
C06218=1204.760,297.936,-68.138,-176.590,7.227,148.364
C06219=1204.756,298.185,-68.168,-176.587,7.230,148.364
C06220=1204.752,298.433,-68.197,-176.585,7.232,148.364
C06221=1204.747,298.681,-68.226,-176.582,7.235,148.364
C06222=1204.743,298.929,-68.256,-176.580,7.237,148.364
C06223=1204.738,299.177,-68.286,-176.577,7.240,148.364
C06224=1204.734,299.426,-68.315,-176.575,7.243,148.364
C06225=1204.730,299.673,-68.345,-176.573,7.245,148.363
C06226=1204.726,299.922,-68.375,-176.570,7.248,148.363
C06227=1204.721,300.170,-68.404,-176.568,7.251,148.363
C06228=1204.717,300.418,-68.434,-176.565,7.254,148.363
C06229=1204.712,300.667,-68.464,-176.563,7.256,148.363
C06230=1204.708,300.915,-68.493,-176.560,7.259,148.363
C06231=1204.704,301.163,-68.523,-176.558,7.262,148.363
C06232=1204.700,301.411,-68.553,-176.556,7.264,148.363
C06233=1204.696,301.659,-68.582,-176.553,7.267,148.363
C06234=1204.691,301.908,-68.612,-176.551,7.269,148.363
C06235=1204.687,302.155,-68.642,-176.548,7.272,148.363
C06236=1204.683,302.404,-68.672,-176.545,7.275,148.363
C06237=1204.679,302.652,-68.701,-176.543,7.278,148.363
C06238=1204.674,302.900,-68.731,-176.541,7.281,148.363
C06239=1204.670,303.148,-68.762,-176.538,7.283,148.363
C06240=1204.666,303.396,-68.791,-176.536,7.286,148.363
C06241=1204.661,303.645,-68.821,-176.533,7.289,148.363
C06242=1204.657,303.893,-68.851,-176.531,7.291,148.363
C06243=1204.653,304.141,-68.881,-176.528,7.294,148.363
C06244=1204.648,304.389,-68.911,-176.526,7.296,148.363
C06245=1204.644,304.637,-68.941,-176.523,7.299,148.363
C06246=1204.640,304.885,-68.970,-176.521,7.302,148.363
C06247=1204.635,305.133,-69.001,-176.519,7.304,148.363
C06248=1204.631,305.382,-69.031,-176.516,7.308,148.363
C06249=1204.627,305.630,-69.060,-176.514,7.310,148.363
C06250=1204.622,305.878,-69.091,-176.512,7.313,148.363
C06251=1204.619,306.127,-69.121,-176.509,7.316,148.363
C06252=1204.615,306.374,-69.151,-176.507,7.318,148.363
C06253=1204.610,306.623,-69.181,-176.504,7.321,148.363
C06254=1204.606,306.871,-69.211,-176.502,7.323,148.363
C06255=1204.601,307.119,-69.241,-176.499,7.326,148.363
C06256=1204.597,307.367,-69.271,-176.497,7.330,148.363
C06257=1204.592,307.615,-69.301,-176.494,7.332,148.363
C06258=1204.588,307.863,-69.331,-176.492,7.335,148.363
C06259=1204.584,308.111,-69.361,-176.490,7.337,148.363
C06260=1204.580,308.359,-69.392,-176.487,7.340,148.363
C06261=1204.575,308.608,-69.421,-176.485,7.343,148.363
C06262=1204.571,308.856,-69.452,-176.483,7.345,148.363
C06263=1204.568,309.104,-69.482,-176.480,7.349,148.363
C06264=1204.563,309.352,-69.512,-176.478,7.351,148.363
C06265=1204.559,309.600,-69.543,-176.475,7.354,148.363
C06266=1204.554,309.848,-69.573,-176.472,7.357,148.363
C06267=1204.550,310.096,-69.603,-176.471,7.359,148.363
C06268=1204.545,310.344,-69.634,-176.468,7.362,148.363
C06269=1204.542,310.593,-69.664,-176.465,7.365,148.363
C06270=1204.537,310.841,-69.694,-176.463,7.368,148.363
C06271=1204.533,311.089,-69.724,-176.460,7.371,148.363
C06272=1204.529,311.337,-69.755,-176.458,7.373,148.363
C06273=1204.524,311.585,-69.785,-176.456,7.376,148.363
C06274=1204.520,311.833,-69.815,-176.453,7.379,148.363
C06275=1204.516,312.082,-69.846,-176.451,7.381,148.363
C06276=1204.512,312.329,-69.877,-176.449,7.384,148.363
C06277=1204.507,312.578,-69.907,-176.446,7.387,148.363
C06278=1204.503,312.826,-69.937,-176.444,7.390,148.363
C06279=1204.499,313.074,-69.968,-176.442,7.393,148.363
C06280=1204.495,313.322,-69.998,-176.439,7.395,148.363
C06281=1204.491,313.570,-70.029,-176.437,7.398,148.363
C06282=1204.486,313.818,-70.059,-176.434,7.401,148.363
C06283=1204.482,314.066,-70.089,-176.432,7.403,148.363
C06284=1204.478,314.315,-70.120,-176.430,7.407,148.363
C06285=1204.473,314.591,-70.154,-176.427,7.410,148.363
C06286=1204.468,314.867,-70.188,-176.424,7.413,148.363
C06287=1204.463,315.143,-70.222,-176.422,7.416,148.363
C06288=1204.458,315.419,-70.256,-176.419,7.419,148.363
C06289=1204.455,315.667,-70.286,-176.416,7.422,148.363
C06290=1204.450,315.915,-70.317,-176.415,7.424,148.363
C06291=1204.446,316.163,-70.348,-176.412,7.427,148.363
C06292=1204.442,316.412,-70.378,-176.409,7.430,148.363
C06293=1204.438,316.660,-70.409,-176.408,7.433,148.363
C06294=1204.433,316.908,-70.440,-176.405,7.436,148.363
C06295=1204.428,317.156,-70.471,-176.402,7.439,148.363
C06296=1204.425,317.404,-70.501,-176.400,7.441,148.363
C06297=1204.421,317.652,-70.532,-176.398,7.445,148.363
C06298=1204.416,317.900,-70.563,-176.395,7.448,148.363
C06299=1204.412,318.149,-70.594,-176.393,7.450,148.363
C06300=1204.408,318.396,-70.624,-176.390,7.453,148.363
C06301=1204.403,318.644,-70.655,-176.389,7.455,148.364
C06302=1204.400,318.892,-70.687,-176.386,7.458,148.364
C06303=1204.395,319.140,-70.718,-176.383,7.461,148.364
C06304=1204.391,319.388,-70.748,-176.382,7.464,148.364
C06305=1204.387,319.636,-70.779,-176.379,7.467,148.364
C06306=1204.383,319.884,-70.810,-176.376,7.470,148.364
C06307=1204.378,320.132,-70.840,-176.375,7.472,148.364
C06308=1204.374,320.381,-70.871,-176.372,7.475,148.364
C06309=1204.370,320.628,-70.902,-176.369,7.478,148.364
C06310=1204.366,320.876,-70.933,-176.368,7.481,148.364
C06311=1204.362,321.125,-70.964,-176.365,7.484,148.364
C06312=1204.357,321.373,-70.995,-176.362,7.487,148.364
C06313=1204.353,321.621,-71.026,-176.361,7.490,148.364
C06314=1204.349,321.869,-71.058,-176.358,7.493,148.364
C06315=1204.344,322.117,-71.088,-176.355,7.496,148.364
C06316=1204.341,322.365,-71.119,-176.354,7.498,148.364
C06317=1204.336,322.613,-71.150,-176.351,7.501,148.364
C06318=1204.332,322.860,-71.181,-176.349,7.504,148.365
C06319=1204.328,323.109,-71.212,-176.347,7.507,148.365
C06320=1204.323,323.357,-71.243,-176.344,7.510,148.365
C06321=1204.320,323.605,-71.275,-176.342,7.512,148.365
C06322=1204.315,323.853,-71.306,-176.340,7.515,148.365
C06323=1204.311,324.101,-71.336,-176.337,7.519,148.365
C06324=1204.307,324.349,-71.368,-176.335,7.521,148.365
C06325=1204.302,324.597,-71.399,-176.333,7.524,148.365
C06326=1204.298,324.845,-71.430,-176.330,7.527,148.365
C06327=1204.294,325.093,-71.462,-176.328,7.529,148.365
C06328=1204.290,325.341,-71.493,-176.326,7.533,148.365
C06329=1204.286,325.589,-71.524,-176.323,7.536,148.365
C06330=1204.282,325.837,-71.555,-176.322,7.538,148.365
C06331=1204.277,326.085,-71.586,-176.319,7.541,148.365
C06332=1204.273,326.333,-71.618,-176.317,7.545,148.366
C06333=1204.269,326.581,-71.649,-176.315,7.547,148.366
C06334=1204.264,326.829,-71.680,-176.312,7.550,148.366
C06335=1204.260,327.077,-71.711,-176.310,7.553,148.366
C06336=1204.256,327.325,-71.743,-176.308,7.556,148.366
C06337=1204.252,327.573,-71.774,-176.305,7.559,148.366
C06338=1204.248,327.821,-71.805,-176.303,7.562,148.366
C06339=1204.244,328.069,-71.837,-176.301,7.564,148.366
C06340=1204.239,328.317,-71.868,-176.299,7.568,148.366
C06341=1204.235,328.565,-71.899,-176.297,7.570,148.366
C06342=1204.231,328.813,-71.931,-176.295,7.573,148.367
C06343=1204.227,329.061,-71.963,-176.292,7.576,148.367
C06344=1204.223,329.309,-71.993,-176.290,7.579,148.367
C06345=1204.219,329.557,-72.025,-176.287,7.582,148.367
C06346=1204.214,329.805,-72.056,-176.285,7.585,148.367
C06347=1204.210,330.053,-72.088,-176.283,7.587,148.367
C06348=1204.206,330.300,-72.120,-176.281,7.591,148.367
C06349=1204.202,330.549,-72.151,-176.278,7.594,148.367
C06350=1204.197,330.796,-72.182,-176.277,7.596,148.367
C06351=1204.194,331.044,-72.214,-176.274,7.599,148.367
C06352=1204.190,331.293,-72.245,-176.272,7.603,148.368
C06353=1204.185,331.541,-72.277,-176.270,7.605,148.368
C06354=1204.181,331.789,-72.309,-176.267,7.608,148.368
C06355=1204.177,332.036,-72.341,-176.265,7.611,148.368
C06356=1204.173,332.285,-72.372,-176.263,7.614,148.368
C06357=1204.168,332.532,-72.403,-176.261,7.617,148.368
C06358=1204.164,332.780,-72.436,-176.259,7.620,148.368
C06359=1204.160,333.029,-72.468,-176.256,7.622,148.368
C06360=1204.155,333.276,-72.498,-176.254,7.626,148.368
C06361=1204.152,333.525,-72.530,-176.252,7.629,148.369
C06362=1204.147,333.772,-72.562,-176.250,7.631,148.369
C06363=1204.143,334.020,-72.594,-176.248,7.635,148.369
C06364=1204.139,334.268,-72.626,-176.245,7.638,148.369
C06365=1204.135,334.516,-72.658,-176.243,7.640,148.369
C06366=1204.130,334.765,-72.689,-176.241,7.644,148.369
C06367=1204.126,335.012,-72.721,-176.238,7.647,148.369
C06368=1204.122,335.260,-72.753,-176.237,7.649,148.369
C06369=1204.119,335.508,-72.784,-176.235,7.652,148.370
C06370=1204.114,335.756,-72.817,-176.233,7.655,148.370
C06371=1204.110,336.004,-72.848,-176.230,7.658,148.370
C06372=1204.106,336.252,-72.880,-176.228,7.661,148.370
C06373=1204.101,336.499,-72.912,-176.226,7.664,148.370
C06374=1204.097,336.747,-72.944,-176.224,7.667,148.370
C06375=1204.094,336.995,-72.976,-176.221,7.670,148.370
C06376=1204.089,337.243,-73.008,-176.220,7.673,148.371
C06377=1204.085,337.491,-73.040,-176.218,7.676,148.371
C06378=1204.081,337.739,-73.072,-176.215,7.679,148.371
C06379=1204.076,337.987,-73.104,-176.213,7.682,148.371
C06380=1204.072,338.235,-73.136,-176.211,7.685,148.371
C06381=1204.068,338.483,-73.168,-176.209,7.688,148.371
C06382=1204.064,338.731,-73.200,-176.207,7.691,148.371
C06383=1204.060,338.979,-73.231,-176.204,7.694,148.372
C06384=1204.056,339.227,-73.264,-176.202,7.697,148.372
C06385=1204.051,339.474,-73.295,-176.201,7.700,148.372
C06386=1204.047,339.723,-73.328,-176.198,7.703,148.372
C06387=1204.043,339.971,-73.360,-176.196,7.706,148.372
C06388=1204.039,340.218,-73.391,-176.194,7.709,148.372
C06389=1204.034,340.497,-73.428,-176.192,7.712,148.373
C06390=1204.029,340.774,-73.464,-176.190,7.715,148.373
C06391=1204.025,341.053,-73.500,-176.187,7.719,148.373
C06392=1204.019,341.331,-73.536,-176.184,7.722,148.373
C06393=1204.016,341.579,-73.568,-176.182,7.725,148.373
C06394=1204.012,341.827,-73.601,-176.180,7.728,148.374
C06395=1204.008,342.075,-73.633,-176.178,7.732,148.374
C06396=1204.003,342.323,-73.665,-176.176,7.734,148.374
C06397=1203.999,342.571,-73.697,-176.174,7.738,148.374
C06398=1203.995,342.819,-73.730,-176.172,7.740,148.374
C06399=1203.991,343.067,-73.762,-176.170,7.743,148.375
C06400=1203.986,343.314,-73.794,-176.168,7.746,148.375
C06401=1203.983,343.562,-73.826,-176.166,7.749,148.375
C06402=1203.978,343.810,-73.859,-176.164,7.752,148.375
C06403=1203.975,344.058,-73.891,-176.161,7.756,148.375
C06404=1203.970,344.306,-73.923,-176.160,7.758,148.375
C06405=1203.965,344.553,-73.956,-176.158,7.761,148.376
C06406=1203.962,344.802,-73.988,-176.155,7.765,148.376
C06407=1203.957,345.050,-74.020,-176.154,7.767,148.376
C06408=1203.954,345.297,-74.053,-176.151,7.771,148.376
C06409=1203.949,345.545,-74.085,-176.149,7.774,148.376
C06410=1203.945,345.793,-74.118,-176.148,7.776,148.377
C06411=1203.941,346.041,-74.150,-176.145,7.780,148.377
C06412=1203.937,346.289,-74.182,-176.144,7.782,148.377
C06413=1203.932,346.537,-74.215,-176.142,7.786,148.377
C06414=1203.929,346.785,-74.247,-176.139,7.789,148.377
C06415=1203.924,347.032,-74.280,-176.138,7.792,148.378
C06416=1203.920,347.280,-74.312,-176.135,7.795,148.378
C06417=1203.916,347.528,-74.345,-176.133,7.798,148.378
C06418=1203.912,347.776,-74.377,-176.132,7.801,148.378
C06419=1203.908,348.024,-74.411,-176.129,7.804,148.379
C06420=1203.904,348.272,-74.442,-176.128,7.807,148.379
C06421=1203.899,348.519,-74.475,-176.125,7.810,148.379
C06422=1203.895,348.767,-74.508,-176.123,7.813,148.379
C06423=1203.891,349.015,-74.540,-176.122,7.816,148.379
C06424=1203.887,349.263,-74.573,-176.119,7.819,148.380
C06425=1203.883,349.511,-74.606,-176.118,7.823,148.380
C06426=1203.879,349.759,-74.638,-176.116,7.825,148.380
C06427=1203.875,350.006,-74.671,-176.114,7.829,148.380
C06428=1203.871,350.254,-74.704,-176.112,7.831,148.381
C06429=1203.866,350.502,-74.736,-176.110,7.834,148.381
C06430=1203.862,350.749,-74.769,-176.108,7.838,148.381
C06431=1203.858,350.998,-74.801,-176.106,7.840,148.381
C06432=1203.854,351.245,-74.834,-176.104,7.844,148.382
C06433=1203.850,351.493,-74.867,-176.102,7.847,148.382
C06434=1203.845,351.741,-74.900,-176.100,7.850,148.382
C06435=1203.842,351.989,-74.932,-176.098,7.853,148.382
C06436=1203.838,352.236,-74.966,-176.096,7.856,148.382
C06437=1203.833,352.485,-74.998,-176.094,7.859,148.383
C06438=1203.829,352.733,-75.031,-176.092,7.863,148.383
C06439=1203.825,352.980,-75.064,-176.091,7.865,148.383
C06440=1203.821,353.228,-75.097,-176.089,7.868,148.384
C06441=1203.817,353.476,-75.129,-176.087,7.871,148.384
C06442=1203.813,353.724,-75.162,-176.085,7.875,148.384
C06443=1203.809,353.972,-75.196,-176.083,7.878,148.384
C06444=1203.804,354.219,-75.228,-176.081,7.880,148.385
C06445=1203.800,354.466,-75.262,-176.079,7.884,148.385
C06446=1203.795,354.715,-75.294,-176.078,7.887,148.385
C06447=1203.792,354.962,-75.327,-176.076,7.890,148.385
C06448=1203.788,355.210,-75.360,-176.073,7.893,148.386
C06449=1203.784,355.458,-75.393,-176.072,7.896,148.386
C06450=1203.780,355.705,-75.426,-176.070,7.899,148.386
C06451=1203.775,355.953,-75.459,-176.068,7.902,148.386
C06452=1203.771,356.201,-75.492,-176.067,7.906,148.387
C06453=1203.767,356.449,-75.525,-176.064,7.909,148.387
C06454=1203.763,356.697,-75.558,-176.063,7.911,148.387
C06455=1203.759,356.945,-75.591,-176.061,7.915,148.388
C06456=1203.754,357.192,-75.624,-176.059,7.918,148.388
C06457=1203.750,357.440,-75.657,-176.057,7.921,148.388
C06458=1203.746,357.688,-75.691,-176.055,7.925,148.389
C06459=1203.742,357.935,-75.724,-176.054,7.927,148.389
C06460=1203.738,358.183,-75.757,-176.052,7.931,148.389
C06461=1203.734,358.432,-75.790,-176.050,7.933,148.389
C06462=1203.731,358.679,-75.823,-176.048,7.937,148.390
C06463=1203.727,358.927,-75.856,-176.047,7.939,148.390
C06464=1203.723,359.174,-75.889,-176.044,7.943,148.390
C06465=1203.719,359.422,-75.922,-176.043,7.946,148.391
C06466=1203.714,359.670,-75.956,-176.041,7.949,148.391
C06467=1203.710,359.918,-75.989,-176.039,7.952,148.391
C06468=1203.705,360.166,-76.022,-176.038,7.955,148.391
C06469=1203.701,360.413,-76.056,-176.036,7.959,148.392
C06470=1203.697,360.661,-76.089,-176.034,7.961,148.392
C06471=1203.693,360.909,-76.122,-176.032,7.965,148.392
C06472=1203.689,361.157,-76.155,-176.031,7.968,148.393
C06473=1203.685,361.404,-76.188,-176.029,7.971,148.393
C06474=1203.681,361.652,-76.221,-176.028,7.974,148.393
C06475=1203.677,361.900,-76.256,-176.026,7.977,148.394
C06476=1203.673,362.148,-76.289,-176.024,7.981,148.394
C06477=1203.669,362.395,-76.322,-176.022,7.983,148.394
C06478=1203.665,362.643,-76.355,-176.020,7.987,148.395
C06479=1203.661,362.891,-76.388,-176.019,7.990,148.395
C06480=1203.657,363.139,-76.421,-176.017,7.993,148.395
C06481=1203.653,363.386,-76.455,-176.016,7.996,148.396
C06482=1203.648,363.634,-76.489,-176.014,7.999,148.396
C06483=1203.644,363.881,-76.522,-176.012,8.002,148.396
C06484=1203.640,364.130,-76.556,-176.011,8.005,148.397
C06485=1203.636,364.377,-76.590,-176.009,8.008,148.397
C06486=1203.632,364.625,-76.623,-176.008,8.011,148.397
C06487=1203.628,364.872,-76.656,-176.006,8.015,148.398
C06488=1203.624,365.120,-76.689,-176.005,8.017,148.398
C06489=1203.620,365.367,-76.723,-176.003,8.021,148.399
C06490=1203.615,365.615,-76.757,-176.001,8.024,148.399
C06491=1203.612,365.864,-76.790,-176.000,8.027,148.399
C06492=1203.608,366.111,-76.824,-175.998,8.030,148.400
C06493=1203.603,366.392,-76.862,-175.997,8.034,148.400
C06494=1203.599,366.672,-76.900,-175.995,8.037,148.401
C06495=1203.594,366.952,-76.938,-175.993,8.041,148.401
C06496=1203.590,367.233,-76.976,-175.991,8.045,148.401
C06497=1203.585,367.481,-77.010,-175.990,8.047,148.402
C06498=1203.581,367.729,-77.043,-175.988,8.050,148.402
C06499=1203.577,367.976,-77.077,-175.987,8.054,148.402
C06500=1203.573,368.224,-77.110,-175.985,8.056,148.403
C06501=1203.568,368.472,-77.144,-175.984,8.060,148.403
C06502=1203.565,368.719,-77.178,-175.982,8.063,148.404
C06503=1203.561,368.967,-77.211,-175.981,8.066,148.404
C06504=1203.557,369.215,-77.245,-175.979,8.069,148.405
C06505=1203.552,369.463,-77.279,-175.978,8.072,148.405
C06506=1203.548,369.710,-77.313,-175.977,8.075,148.405
C06507=1203.544,369.957,-77.346,-175.975,8.079,148.406
C06508=1203.540,370.206,-77.381,-175.974,8.081,148.406
C06509=1203.536,370.453,-77.414,-175.973,8.084,148.407
C06510=1203.532,370.700,-77.448,-175.971,8.088,148.407
C06511=1203.527,370.948,-77.481,-175.970,8.091,148.407
C06512=1203.524,371.196,-77.516,-175.969,8.093,148.408
C06513=1203.520,371.444,-77.549,-175.967,8.097,148.408
C06514=1203.516,371.691,-77.583,-175.966,8.100,148.409
C06515=1203.511,371.939,-77.616,-175.964,8.103,148.409
C06516=1203.508,372.187,-77.651,-175.963,8.105,148.409
C06517=1203.503,372.435,-77.684,-175.961,8.109,148.410
C06518=1203.499,372.682,-77.718,-175.960,8.112,148.410
C06519=1203.496,372.929,-77.752,-175.959,8.115,148.411
C06520=1203.491,373.178,-77.786,-175.958,8.118,148.411
C06521=1203.488,373.425,-77.820,-175.956,8.121,148.411
C06522=1203.483,373.673,-77.853,-175.955,8.124,148.412
C06523=1203.479,373.920,-77.888,-175.954,8.127,148.412
C06524=1203.476,374.168,-77.922,-175.953,8.130,148.413
C06525=1203.471,374.416,-77.956,-175.951,8.134,148.413
C06526=1203.467,374.663,-77.990,-175.950,8.136,148.414
C06527=1203.464,374.911,-78.024,-175.949,8.139,148.414
C06528=1203.459,375.159,-78.058,-175.947,8.142,148.414
C06529=1203.455,375.406,-78.092,-175.947,8.145,148.415
C06530=1203.450,375.654,-78.126,-175.945,8.148,148.415
C06531=1203.447,375.902,-78.160,-175.944,8.151,148.416
C06532=1203.442,376.149,-78.194,-175.942,8.154,148.416
C06533=1203.438,376.396,-78.228,-175.942,8.157,148.417
C06534=1203.435,376.644,-78.262,-175.940,8.160,148.417
C06535=1203.430,376.892,-78.296,-175.939,8.163,148.418
C06536=1203.426,377.139,-78.330,-175.938,8.166,148.418
C06537=1203.423,377.388,-78.365,-175.937,8.169,148.419
C06538=1203.419,377.635,-78.398,-175.936,8.173,148.419
C06539=1203.414,377.883,-78.432,-175.934,8.175,148.419
C06540=1203.411,378.131,-78.466,-175.934,8.178,148.420
C06541=1203.406,378.378,-78.501,-175.932,8.181,148.420
C06542=1203.402,378.625,-78.535,-175.931,8.184,148.421
C06543=1203.398,378.873,-78.570,-175.930,8.187,148.421
C06544=1203.394,379.121,-78.603,-175.929,8.190,148.422
C06545=1203.390,379.368,-78.637,-175.928,8.193,148.422
C06546=1203.386,379.616,-78.671,-175.927,8.196,148.423
C06547=1203.382,379.864,-78.706,-175.926,8.199,148.423
C06548=1203.378,380.111,-78.740,-175.925,8.202,148.424
C06549=1203.374,380.359,-78.775,-175.924,8.205,148.424
C06550=1203.370,380.606,-78.808,-175.923,8.207,148.424
C06551=1203.366,380.855,-78.843,-175.922,8.211,148.425
C06552=1203.361,381.102,-78.877,-175.921,8.213,148.425
C06553=1203.357,381.349,-78.911,-175.920,8.216,148.426
C06554=1203.353,381.597,-78.946,-175.919,8.219,148.426
C06555=1203.350,381.844,-78.980,-175.918,8.222,148.427
C06556=1203.345,382.092,-79.014,-175.917,8.225,148.427
C06557=1203.342,382.340,-79.048,-175.916,8.228,148.428
C06558=1203.337,382.587,-79.083,-175.915,8.231,148.428
C06559=1203.333,382.835,-79.118,-175.914,8.234,148.429
C06560=1203.329,383.082,-79.152,-175.913,8.237,148.429
C06561=1203.325,383.330,-79.186,-175.912,8.240,148.430
C06562=1203.321,383.578,-79.220,-175.911,8.242,148.430
C06563=1203.317,383.826,-79.254,-175.911,8.245,148.431
C06564=1203.313,384.074,-79.289,-175.909,8.248,148.431
C06565=1203.309,384.321,-79.323,-175.909,8.251,148.432
C06566=1203.304,384.568,-79.357,-175.908,8.254,148.432
C06567=1203.301,384.816,-79.391,-175.907,8.257,148.433
C06568=1203.297,385.063,-79.426,-175.906,8.260,148.433
C06569=1203.293,385.312,-79.461,-175.905,8.262,148.434
C06570=1203.289,385.558,-79.495,-175.904,8.265,148.434
C06571=1203.285,385.805,-79.530,-175.904,8.268,148.435
C06572=1203.281,386.054,-79.565,-175.902,8.271,148.435
C06573=1203.277,386.301,-79.598,-175.902,8.274,148.436
C06574=1203.273,386.549,-79.633,-175.901,8.276,148.436
C06575=1203.268,386.796,-79.668,-175.900,8.279,148.437
C06576=1203.265,387.044,-79.702,-175.899,8.282,148.437
C06577=1203.260,387.291,-79.736,-175.898,8.285,148.438
C06578=1203.256,387.540,-79.771,-175.898,8.287,148.438
C06579=1203.253,387.787,-79.805,-175.897,8.291,148.439
C06580=1203.248,388.034,-79.840,-175.896,8.293,148.439
C06581=1203.244,388.282,-79.874,-175.895,8.296,148.440
C06582=1203.241,388.529,-79.909,-175.895,8.299,148.441
C06583=1203.237,388.777,-79.944,-175.894,8.302,148.441
C06584=1203.232,389.024,-79.978,-175.893,8.305,148.441
C06585=1203.228,389.272,-80.013,-175.893,8.307,148.442
C06586=1203.224,389.519,-80.047,-175.892,8.310,148.443
C06587=1203.220,389.768,-80.082,-175.891,8.313,148.443
C06588=1203.216,390.015,-80.116,-175.891,8.315,148.444
C06589=1203.213,390.262,-80.151,-175.890,8.318,148.444
C06590=1203.208,390.510,-80.186,-175.889,8.321,148.445
C06591=1203.204,390.758,-80.221,-175.888,8.323,148.445
C06592=1203.200,391.005,-80.255,-175.888,8.326,148.446
C06593=1203.196,391.253,-80.289,-175.887,8.329,148.446
C06594=1203.192,391.500,-80.324,-175.887,8.332,148.447
C06595=1203.188,391.748,-80.359,-175.886,8.334,148.447
C06596=1203.184,391.995,-80.394,-175.885,8.337,148.448
C06597=1203.179,392.278,-80.434,-175.884,8.340,148.448
C06598=1203.175,392.561,-80.473,-175.884,8.343,148.449
C06599=1203.170,392.843,-80.513,-175.883,8.346,148.449
C06600=1203.165,393.126,-80.552,-175.882,8.349,148.450
C06601=1203.162,393.374,-80.586,-175.882,8.352,148.451
C06602=1203.158,393.621,-80.622,-175.881,8.355,148.451
C06603=1203.154,393.869,-80.656,-175.881,8.357,148.452
C06604=1203.149,394.116,-80.691,-175.880,8.360,148.452
C06605=1203.145,394.364,-80.726,-175.880,8.362,148.453
C06606=1203.142,394.611,-80.760,-175.879,8.365,148.453
C06607=1203.138,394.859,-80.795,-175.879,8.367,148.454
C06608=1203.133,395.107,-80.830,-175.878,8.370,148.454
C06609=1203.129,395.354,-80.865,-175.877,8.372,148.455
C06610=1203.125,395.601,-80.900,-175.877,8.375,148.455
C06611=1203.122,395.849,-80.934,-175.876,8.378,148.456
C06612=1203.117,396.096,-80.969,-175.876,8.380,148.456
C06613=1203.113,396.344,-81.004,-175.875,8.383,148.457
C06614=1203.109,396.592,-81.038,-175.875,8.385,148.457
C06615=1203.105,396.839,-81.074,-175.874,8.387,148.458
C06616=1203.101,397.087,-81.108,-175.873,8.391,148.458
C06617=1203.098,397.334,-81.143,-175.873,8.393,148.459
C06618=1203.094,397.582,-81.178,-175.873,8.395,148.459
C06619=1203.089,397.829,-81.213,-175.872,8.398,148.460
C06620=1203.085,398.077,-81.248,-175.872,8.400,148.461
C06621=1203.081,398.324,-81.283,-175.871,8.402,148.461
C06622=1203.077,398.572,-81.317,-175.871,8.405,148.462
C06623=1203.073,398.819,-81.353,-175.870,8.408,148.462
C06624=1203.069,399.067,-81.388,-175.870,8.410,148.463
C06625=1203.065,399.314,-81.422,-175.869,8.413,148.463
C06626=1203.061,399.562,-81.457,-175.869,8.415,148.464
C06627=1203.057,399.809,-81.492,-175.868,8.417,148.464
C06628=1203.053,400.057,-81.527,-175.868,8.420,148.465
C06629=1203.049,400.305,-81.562,-175.867,8.423,148.465
C06630=1203.045,400.552,-81.597,-175.867,8.425,148.466
C06631=1203.041,400.800,-81.632,-175.867,8.427,148.466
C06632=1203.036,401.047,-81.667,-175.866,8.430,148.467
C06633=1203.032,401.295,-81.702,-175.866,8.433,148.467
C06634=1203.029,401.542,-81.737,-175.865,8.435,148.468
C06635=1203.025,401.789,-81.771,-175.865,8.437,148.468
C06636=1203.021,402.037,-81.807,-175.864,8.440,148.469
C06637=1203.017,402.284,-81.841,-175.864,8.442,148.469
C06638=1203.013,402.532,-81.877,-175.864,8.445,148.470
C06639=1203.009,402.780,-81.912,-175.864,8.447,148.470
C06640=1203.005,403.027,-81.947,-175.863,8.449,148.471
C06641=1203.001,403.275,-81.982,-175.862,8.452,148.471
C06642=1202.997,403.522,-82.017,-175.862,8.454,148.472
C06643=1202.993,403.770,-82.052,-175.862,8.456,148.472
C06644=1202.989,404.017,-82.087,-175.862,8.459,148.473
C06645=1202.984,404.265,-82.122,-175.861,8.461,148.473
C06646=1202.981,404.512,-82.157,-175.861,8.463,148.474
C06647=1202.976,404.760,-82.192,-175.860,8.465,148.474
C06648=1202.973,405.007,-82.227,-175.860,8.468,148.475
C06649=1202.969,405.255,-82.262,-175.859,8.471,148.475
C06650=1202.964,405.502,-82.297,-175.859,8.473,148.476
C06651=1202.960,405.750,-82.332,-175.859,8.475,148.477
C06652=1202.956,405.997,-82.367,-175.859,8.477,148.477
C06653=1202.952,406.244,-82.403,-175.859,8.480,148.478
C06654=1202.948,406.493,-82.438,-175.858,8.482,148.478
C06655=1202.944,406.739,-82.473,-175.858,8.484,148.478
C06656=1202.940,406.987,-82.508,-175.857,8.486,148.479
C06657=1202.937,407.235,-82.543,-175.857,8.488,148.480
C06658=1202.932,407.482,-82.578,-175.856,8.492,148.480
C06659=1202.928,407.730,-82.613,-175.856,8.494,148.481
C06660=1202.924,407.977,-82.648,-175.856,8.496,148.481
C06661=1202.920,408.225,-82.683,-175.855,8.498,148.481
C06662=1202.916,408.472,-82.719,-175.855,8.500,148.482
C06663=1202.912,408.719,-82.754,-175.855,8.503,148.483
C06664=1202.908,408.967,-82.789,-175.855,8.505,148.483
C06665=1202.904,409.215,-82.824,-175.854,8.507,148.483
C06666=1202.900,409.461,-82.860,-175.854,8.509,148.484
C06667=1202.896,409.710,-82.894,-175.854,8.511,148.484
C06668=1202.893,409.957,-82.930,-175.853,8.514,148.485
C06669=1202.888,410.205,-82.964,-175.853,8.516,148.486
C06670=1202.884,410.452,-83.000,-175.853,8.518,148.486
C06671=1202.881,410.700,-83.035,-175.852,8.520,148.486
C06672=1202.876,410.947,-83.070,-175.852,8.522,148.487
C06673=1202.872,411.194,-83.105,-175.852,8.525,148.487
C06674=1202.869,411.442,-83.141,-175.851,8.527,148.488
C06675=1202.864,411.689,-83.175,-175.851,8.529,148.489
C06676=1202.861,411.937,-83.211,-175.851,8.531,148.489
C06677=1202.857,412.184,-83.247,-175.850,8.533,148.489
C06678=1202.853,412.431,-83.282,-175.850,8.536,148.490
C06679=1202.849,412.679,-83.317,-175.850,8.538,148.490
C06680=1202.845,412.927,-83.352,-175.850,8.539,148.491
C06681=1202.841,413.174,-83.387,-175.850,8.541,148.491
C06682=1202.837,413.422,-83.422,-175.849,8.544,148.492
C06683=1202.833,413.669,-83.458,-175.849,8.546,148.492
C06684=1202.829,413.916,-83.493,-175.849,8.548,148.493
C06685=1202.824,414.164,-83.529,-175.848,8.550,148.493
C06686=1202.820,414.412,-83.564,-175.848,8.552,148.494
C06687=1202.816,414.659,-83.599,-175.848,8.555,148.494
C06688=1202.813,414.906,-83.635,-175.848,8.557,148.495
C06689=1202.809,415.154,-83.670,-175.847,8.559,148.495
C06690=1202.804,415.401,-83.705,-175.847,8.561,148.496
C06691=1202.801,415.649,-83.740,-175.847,8.563,148.496
C06692=1202.797,415.896,-83.776,-175.847,8.565,148.497
C06693=1202.792,416.197,-83.818,-175.846,8.568,148.497
C06694=1202.788,416.498,-83.862,-175.846,8.570,148.498
C06695=1202.787,416.798,-83.904,-175.845,8.572,148.498
C06696=1202.789,417.099,-83.946,-175.845,8.575,148.499
C06697=1202.367,417.099,-83.984,-175.848,8.585,148.503
C06698=1202.365,416.796,-83.942,-175.849,8.583,148.502
C06699=1202.366,416.493,-83.899,-175.849,8.581,148.501
C06700=1202.371,416.189,-83.855,-175.849,8.579,148.501
C06701=1202.375,415.885,-83.812,-175.850,8.575,148.500
C06702=1202.379,415.638,-83.777,-175.850,8.573,148.500
C06703=1202.383,415.390,-83.742,-175.850,8.572,148.499
C06704=1202.387,415.143,-83.706,-175.850,8.570,148.499
C06705=1202.391,414.895,-83.671,-175.850,8.567,148.498
C06706=1202.394,414.648,-83.635,-175.851,8.565,148.498
C06707=1202.399,414.401,-83.600,-175.851,8.563,148.497
C06708=1202.403,414.153,-83.565,-175.851,8.561,148.497
C06709=1202.407,413.905,-83.529,-175.852,8.558,148.496
C06710=1202.411,413.658,-83.494,-175.852,8.557,148.496
C06711=1202.415,413.410,-83.459,-175.853,8.554,148.495
C06712=1202.419,413.163,-83.424,-175.853,8.552,148.495
C06713=1202.423,412.916,-83.388,-175.852,8.551,148.494
C06714=1202.427,412.669,-83.353,-175.853,8.548,148.494
C06715=1202.431,412.420,-83.318,-175.853,8.546,148.494
C06716=1202.435,412.174,-83.283,-175.854,8.544,148.493
C06717=1202.439,411.926,-83.247,-175.854,8.542,148.493
C06718=1202.443,411.678,-83.213,-175.854,8.540,148.492
C06719=1202.447,411.431,-83.177,-175.854,8.537,148.491
C06720=1202.451,411.184,-83.142,-175.855,8.535,148.491
C06721=1202.454,410.936,-83.106,-175.855,8.533,148.491
C06722=1202.460,410.688,-83.071,-175.855,8.531,148.490
C06723=1202.463,410.441,-83.036,-175.856,8.528,148.490
C06724=1202.467,410.193,-83.000,-175.856,8.526,148.489
C06725=1202.472,409.946,-82.966,-175.857,8.524,148.489
C06726=1202.475,409.699,-82.930,-175.857,8.522,148.488
C06727=1202.479,409.451,-82.895,-175.857,8.520,148.488
C06728=1202.483,409.204,-82.860,-175.857,8.517,148.487
C06729=1202.487,408.956,-82.825,-175.857,8.515,148.487
C06730=1202.491,408.709,-82.789,-175.858,8.513,148.486
C06731=1202.495,408.461,-82.755,-175.858,8.511,148.486
C06732=1202.499,408.214,-82.719,-175.859,8.509,148.485
C06733=1202.503,407.966,-82.684,-175.859,8.506,148.485
C06734=1202.507,407.719,-82.649,-175.859,8.504,148.484
C06735=1202.511,407.471,-82.613,-175.859,8.502,148.484
C06736=1202.515,407.224,-82.579,-175.859,8.500,148.483
C06737=1202.519,406.976,-82.543,-175.860,8.498,148.483
C06738=1202.523,406.728,-82.509,-175.860,8.495,148.482
C06739=1202.527,406.481,-82.473,-175.861,8.492,148.482
C06740=1202.531,406.234,-82.438,-175.861,8.490,148.481
C06741=1202.535,405.986,-82.403,-175.862,8.488,148.481
C06742=1202.539,405.739,-82.368,-175.862,8.485,148.480
C06743=1202.543,405.491,-82.333,-175.862,8.483,148.479
C06744=1202.547,405.243,-82.297,-175.863,8.481,148.479
C06745=1202.551,404.996,-82.263,-175.863,8.479,148.479
C06746=1202.555,404.748,-82.227,-175.863,8.477,148.478
C06747=1202.559,404.502,-82.192,-175.863,8.474,148.478
C06748=1202.563,404.254,-82.157,-175.864,8.471,148.477
C06749=1202.566,404.006,-82.122,-175.864,8.469,148.476
C06750=1202.571,403.759,-82.088,-175.865,8.467,148.476
C06751=1202.575,403.511,-82.052,-175.865,8.465,148.476
C06752=1202.579,403.264,-82.018,-175.866,8.463,148.475
C06753=1202.583,403.017,-81.982,-175.866,8.460,148.475
C06754=1202.587,402.768,-81.948,-175.867,8.457,148.474
C06755=1202.591,402.522,-81.912,-175.867,8.455,148.473
C06756=1202.595,402.274,-81.878,-175.867,8.453,148.473
C06757=1202.599,402.027,-81.842,-175.867,8.450,148.472
C06758=1202.603,401.779,-81.808,-175.868,8.448,148.472
C06759=1202.607,401.531,-81.772,-175.869,8.445,148.471
C06760=1202.611,401.284,-81.738,-175.869,8.443,148.471
C06761=1202.615,401.036,-81.702,-175.869,8.441,148.470
C06762=1202.620,400.789,-81.668,-175.869,8.438,148.470
C06763=1202.623,400.541,-81.632,-175.870,8.435,148.469
C06764=1202.627,400.294,-81.598,-175.870,8.433,148.469
C06765=1202.631,400.047,-81.563,-175.871,8.431,148.468
C06766=1202.635,399.799,-81.528,-175.871,8.429,148.468
C06767=1202.639,399.551,-81.493,-175.872,8.426,148.467
C06768=1202.643,399.304,-81.458,-175.872,8.423,148.467
C06769=1202.648,399.056,-81.423,-175.872,8.421,148.466
C06770=1202.651,398.809,-81.388,-175.873,8.418,148.466
C06771=1202.656,398.561,-81.353,-175.873,8.416,148.465
C06772=1202.659,398.314,-81.318,-175.874,8.414,148.465
C06773=1202.663,398.066,-81.283,-175.875,8.411,148.464
C06774=1202.667,397.819,-81.249,-175.875,8.409,148.464
C06775=1202.671,397.571,-81.213,-175.875,8.406,148.463
C06776=1202.676,397.324,-81.179,-175.876,8.403,148.462
C06777=1202.680,397.075,-81.144,-175.876,8.401,148.462
C06778=1202.684,396.829,-81.109,-175.876,8.399,148.461
C06779=1202.688,396.581,-81.074,-175.878,8.396,148.461
C06780=1202.691,396.334,-81.040,-175.878,8.394,148.460
C06781=1202.695,396.086,-81.005,-175.879,8.390,148.460
C06782=1202.700,395.839,-80.970,-175.879,8.388,148.459
C06783=1202.703,395.591,-80.935,-175.879,8.386,148.459
C06784=1202.707,395.343,-80.900,-175.880,8.383,148.458
C06785=1202.712,395.095,-80.865,-175.881,8.381,148.458
C06786=1202.716,394.848,-80.830,-175.881,8.378,148.457
C06787=1202.719,394.601,-80.796,-175.882,8.375,148.457
C06788=1202.723,394.353,-80.761,-175.882,8.372,148.456
C06789=1202.728,394.105,-80.727,-175.883,8.370,148.456
C06790=1202.732,393.858,-80.691,-175.884,8.367,148.455
C06791=1202.736,393.610,-80.657,-175.884,8.365,148.455
C06792=1202.739,393.363,-80.622,-175.885,8.362,148.454
C06793=1202.744,393.116,-80.587,-175.885,8.360,148.454
C06794=1202.748,392.833,-80.548,-175.886,8.357,148.453
C06795=1202.753,392.550,-80.508,-175.887,8.353,148.452
C06796=1202.758,392.267,-80.469,-175.887,8.350,148.452
C06797=1202.762,391.985,-80.429,-175.888,8.347,148.451
C06798=1202.766,391.737,-80.394,-175.888,8.345,148.451
C06799=1202.771,391.489,-80.360,-175.889,8.342,148.450
C06800=1202.774,391.242,-80.325,-175.890,8.340,148.450
C06801=1202.778,390.995,-80.290,-175.891,8.337,148.449
C06802=1202.782,390.747,-80.255,-175.891,8.334,148.449
C06803=1202.787,390.499,-80.221,-175.892,8.331,148.448
C06804=1202.790,390.251,-80.187,-175.893,8.329,148.448
C06805=1202.795,390.004,-80.152,-175.893,8.326,148.447
C06806=1202.798,389.756,-80.117,-175.894,8.323,148.447
C06807=1202.802,389.509,-80.083,-175.895,8.320,148.446
C06808=1202.806,389.261,-80.048,-175.895,8.318,148.446
C06809=1202.811,389.014,-80.013,-175.896,8.315,148.445
C06810=1202.815,388.766,-79.979,-175.897,8.312,148.444
C06811=1202.818,388.519,-79.945,-175.897,8.310,148.444
C06812=1202.822,388.271,-79.909,-175.898,8.307,148.443
C06813=1202.827,388.024,-79.875,-175.899,8.304,148.443
C06814=1202.830,387.777,-79.841,-175.899,8.301,148.442
C06815=1202.834,387.528,-79.806,-175.900,8.299,148.442
C06816=1202.839,387.281,-79.771,-175.901,8.296,148.441
C06817=1202.843,387.033,-79.737,-175.902,8.292,148.441
C06818=1202.847,386.786,-79.703,-175.903,8.290,148.440
C06819=1202.851,386.538,-79.668,-175.903,8.287,148.440
C06820=1202.855,386.290,-79.633,-175.904,8.284,148.439
C06821=1202.859,386.042,-79.599,-175.905,8.281,148.439
C06822=1202.863,385.796,-79.564,-175.906,8.278,148.438
C06823=1202.867,385.548,-79.530,-175.907,8.276,148.438
C06824=1202.871,385.300,-79.495,-175.908,8.273,148.437
C06825=1202.875,385.053,-79.461,-175.908,8.270,148.437
C06826=1202.878,384.805,-79.427,-175.910,8.267,148.436
C06827=1202.883,384.558,-79.392,-175.910,8.264,148.436
C06828=1202.887,384.310,-79.357,-175.912,8.261,148.435
C06829=1202.891,384.063,-79.323,-175.912,8.259,148.435
C06830=1202.895,383.815,-79.289,-175.912,8.256,148.434
C06831=1202.899,383.567,-79.254,-175.914,8.253,148.434
C06832=1202.903,383.320,-79.220,-175.914,8.250,148.433
C06833=1202.907,383.072,-79.185,-175.916,8.247,148.433
C06834=1202.911,382.825,-79.152,-175.916,8.244,148.432
C06835=1202.916,382.577,-79.117,-175.918,8.241,148.432
C06836=1202.920,382.329,-79.082,-175.918,8.238,148.431
C06837=1202.923,382.082,-79.048,-175.920,8.236,148.431
C06838=1202.928,381.833,-79.014,-175.920,8.232,148.430
C06839=1202.931,381.586,-78.980,-175.922,8.230,148.430
C06840=1202.936,381.339,-78.946,-175.922,8.227,148.429
C06841=1202.939,381.091,-78.912,-175.924,8.224,148.429
C06842=1202.944,380.843,-78.877,-175.924,8.221,148.428
C06843=1202.948,380.596,-78.843,-175.926,8.218,148.428
C06844=1202.952,380.348,-78.809,-175.926,8.215,148.427
C06845=1202.956,380.101,-78.774,-175.928,8.212,148.427
C06846=1202.959,379.853,-78.740,-175.929,8.209,148.427
C06847=1202.964,379.605,-78.706,-175.930,8.206,148.426
C06848=1202.968,379.358,-78.672,-175.931,8.203,148.426
C06849=1202.972,379.110,-78.637,-175.932,8.200,148.425
C06850=1202.976,378.863,-78.604,-175.933,8.197,148.425
C06851=1202.981,378.615,-78.569,-175.934,8.194,148.424
C06852=1202.984,378.367,-78.535,-175.935,8.191,148.424
C06853=1202.989,378.119,-78.501,-175.936,8.189,148.423
C06854=1202.992,377.872,-78.467,-175.937,8.186,148.423
C06855=1202.996,377.624,-78.432,-175.938,8.183,148.422
C06856=1203.000,377.377,-78.399,-175.939,8.180,148.422
C06857=1203.005,377.130,-78.364,-175.940,8.177,148.422
C06858=1203.008,376.881,-78.331,-175.942,8.173,148.421
C06859=1203.013,376.634,-78.296,-175.943,8.170,148.420
C06860=1203.017,376.387,-78.262,-175.944,8.167,148.420
C06861=1203.021,376.138,-78.228,-175.945,8.165,148.420
C06862=1203.025,375.891,-78.194,-175.946,8.162,148.419
C06863=1203.029,375.643,-78.160,-175.947,8.159,148.419
C06864=1203.033,375.396,-78.126,-175.949,8.155,148.418
C06865=1203.037,375.148,-78.092,-175.950,8.152,148.418
C06866=1203.041,374.900,-78.058,-175.951,8.149,148.417
C06867=1203.045,374.653,-78.024,-175.952,8.146,148.417
C06868=1203.050,374.405,-77.990,-175.954,8.144,148.417
C06869=1203.053,374.157,-77.956,-175.955,8.140,148.416
C06870=1203.057,373.910,-77.922,-175.957,8.137,148.416
C06871=1203.061,373.662,-77.888,-175.958,8.134,148.415
C06872=1203.065,373.415,-77.854,-175.958,8.131,148.415
C06873=1203.070,373.167,-77.820,-175.960,8.128,148.414
C06874=1203.074,372.919,-77.787,-175.961,8.125,148.414
C06875=1203.077,372.672,-77.752,-175.963,8.122,148.414
C06876=1203.082,372.424,-77.719,-175.964,8.119,148.413
C06877=1203.086,372.176,-77.685,-175.966,8.116,148.413
C06878=1203.090,371.929,-77.651,-175.967,8.113,148.412
C06879=1203.094,371.681,-77.617,-175.968,8.110,148.412
C06880=1203.098,371.433,-77.583,-175.969,8.107,148.412
C06881=1203.102,371.186,-77.550,-175.971,8.103,148.411
C06882=1203.107,370.938,-77.515,-175.972,8.101,148.411
C06883=1203.110,370.690,-77.482,-175.974,8.098,148.410
C06884=1203.114,370.443,-77.448,-175.975,8.094,148.410
C06885=1203.119,370.195,-77.414,-175.976,8.091,148.409
C06886=1203.123,369.948,-77.380,-175.978,8.089,148.409
C06887=1203.126,369.699,-77.347,-175.979,8.085,148.409
C06888=1203.131,369.452,-77.312,-175.981,8.082,148.408
C06889=1203.135,369.204,-77.279,-175.982,8.079,148.408
C06890=1203.139,368.957,-77.245,-175.984,8.076,148.407
C06891=1203.143,368.709,-77.212,-175.985,8.073,148.407
C06892=1203.147,368.460,-77.178,-175.986,8.070,148.407
C06893=1203.151,368.213,-77.144,-175.988,8.066,148.406
C06894=1203.155,367.966,-77.111,-175.989,8.064,148.406
C06895=1203.159,367.719,-77.077,-175.991,8.060,148.405
C06896=1203.164,367.470,-77.043,-175.993,8.057,148.405
C06897=1203.167,367.222,-77.010,-175.994,8.055,148.405
C06898=1203.173,366.942,-76.972,-175.995,8.051,148.404
C06899=1203.177,366.662,-76.934,-175.997,8.047,148.404
C06900=1203.181,366.381,-76.895,-175.999,8.044,148.403
C06901=1203.186,366.100,-76.858,-176.001,8.040,148.403
C06902=1203.190,365.853,-76.824,-176.002,8.037,148.403
C06903=1203.194,365.605,-76.790,-176.004,8.034,148.402
C06904=1203.198,365.357,-76.757,-176.005,8.031,148.402
C06905=1203.202,365.110,-76.723,-176.007,8.028,148.402
C06906=1203.206,364.862,-76.690,-176.008,8.025,148.401
C06907=1203.211,364.614,-76.656,-176.010,8.021,148.401
C06908=1203.215,364.367,-76.622,-176.012,8.019,148.401
C06909=1203.219,364.119,-76.589,-176.014,8.015,148.400
C06910=1203.222,363.871,-76.556,-176.015,8.012,148.400
C06911=1203.226,363.623,-76.522,-176.017,8.009,148.400
C06912=1203.231,363.375,-76.489,-176.018,8.006,148.399
C06913=1203.234,363.128,-76.455,-176.020,8.002,148.399
C06914=1203.239,362.880,-76.422,-176.022,8.000,148.399
C06915=1203.243,362.633,-76.389,-176.023,7.996,148.398
C06916=1203.248,362.384,-76.355,-176.025,7.993,148.398
C06917=1203.252,362.137,-76.322,-176.027,7.990,148.397
C06918=1203.255,361.889,-76.288,-176.028,7.987,148.397
C06919=1203.259,361.641,-76.255,-176.030,7.984,148.397
C06920=1203.263,361.393,-76.222,-176.032,7.981,148.396
C06921=1203.267,361.146,-76.188,-176.034,7.978,148.396
C06922=1203.272,360.898,-76.155,-176.035,7.975,148.396
C06923=1203.276,360.650,-76.122,-176.037,7.971,148.395
C06924=1203.280,360.403,-76.089,-176.038,7.969,148.395
C06925=1203.284,360.155,-76.056,-176.040,7.965,148.395
C06926=1203.288,359.907,-76.023,-176.042,7.962,148.395
C06927=1203.292,359.659,-75.990,-176.044,7.959,148.394
C06928=1203.296,359.412,-75.956,-176.046,7.956,148.394
C06929=1203.300,359.165,-75.923,-176.047,7.953,148.394
C06930=1203.304,358.917,-75.889,-176.049,7.949,148.393
C06931=1203.308,358.668,-75.856,-176.050,7.947,148.393
C06932=1203.312,358.421,-75.823,-176.053,7.943,148.393
C06933=1203.316,358.173,-75.790,-176.055,7.940,148.392
C06934=1203.320,357.925,-75.756,-176.056,7.937,148.392
C06935=1203.325,357.677,-75.724,-176.058,7.934,148.392
C06936=1203.329,357.429,-75.691,-176.060,7.931,148.391
C06937=1203.333,357.181,-75.658,-176.062,7.928,148.391
C06938=1203.337,356.934,-75.624,-176.064,7.924,148.391
C06939=1203.341,356.686,-75.591,-176.065,7.922,148.391
C06940=1203.345,356.438,-75.558,-176.067,7.918,148.390
C06941=1203.350,356.190,-75.525,-176.069,7.916,148.390
C06942=1203.354,355.943,-75.492,-176.071,7.912,148.390
C06943=1203.358,355.695,-75.459,-176.073,7.909,148.390
C06944=1203.362,355.447,-75.426,-176.075,7.906,148.389
C06945=1203.366,355.199,-75.394,-176.076,7.903,148.389
C06946=1203.370,354.952,-75.361,-176.078,7.900,148.389
C06947=1203.374,354.704,-75.327,-176.080,7.897,148.388
C06948=1203.378,354.456,-75.294,-176.082,7.893,148.388
C06949=1203.382,354.208,-75.261,-176.084,7.891,148.388
C06950=1203.386,353.961,-75.228,-176.086,7.887,148.388
C06951=1203.391,353.712,-75.195,-176.088,7.885,148.387
C06952=1203.395,353.465,-75.162,-176.089,7.881,148.387
C06953=1203.399,353.218,-75.130,-176.092,7.878,148.387
C06954=1203.403,352.970,-75.097,-176.093,7.875,148.387
C06955=1203.408,352.722,-75.065,-176.096,7.872,148.386
C06956=1203.412,352.474,-75.031,-176.097,7.868,148.386
C06957=1203.416,352.226,-74.998,-176.099,7.866,148.386
C06958=1203.420,351.978,-74.966,-176.101,7.862,148.386
C06959=1203.424,351.731,-74.933,-176.103,7.860,148.385
C06960=1203.428,351.483,-74.900,-176.105,7.857,148.385
C06961=1203.432,351.235,-74.867,-176.107,7.853,148.385
C06962=1203.436,350.987,-74.834,-176.108,7.850,148.385
C06963=1203.440,350.739,-74.802,-176.111,7.847,148.384
C06964=1203.444,350.491,-74.769,-176.113,7.844,148.384
C06965=1203.448,350.243,-74.736,-176.115,7.841,148.384
C06966=1203.453,349.996,-74.703,-176.117,7.838,148.384
C06967=1203.457,349.748,-74.672,-176.118,7.835,148.384
C06968=1203.461,349.500,-74.638,-176.120,7.832,148.383
C06969=1203.465,349.252,-74.606,-176.122,7.828,148.383
C06970=1203.470,349.004,-74.573,-176.124,7.826,148.383
C06971=1203.473,348.757,-74.540,-176.126,7.823,148.382
C06972=1203.477,348.509,-74.508,-176.129,7.819,148.382
C06973=1203.481,348.261,-74.475,-176.130,7.817,148.382
C06974=1203.486,348.014,-74.443,-176.132,7.813,148.382
C06975=1203.490,347.766,-74.410,-176.134,7.811,148.382
C06976=1203.494,347.517,-74.378,-176.136,7.807,148.381
C06977=1203.498,347.270,-74.345,-176.139,7.804,148.381
C06978=1203.502,347.022,-74.313,-176.140,7.802,148.381
C06979=1203.506,346.774,-74.280,-176.142,7.798,148.381
C06980=1203.510,346.526,-74.248,-176.145,7.795,148.381
C06981=1203.515,346.278,-74.216,-176.146,7.792,148.380
C06982=1203.519,346.031,-74.182,-176.149,7.789,148.380
C06983=1203.523,345.782,-74.151,-176.151,7.786,148.380
C06984=1203.527,345.535,-74.117,-176.152,7.783,148.380
C06985=1203.532,345.286,-74.085,-176.155,7.780,148.380
C06986=1203.536,345.039,-74.054,-176.157,7.777,148.379
C06987=1203.540,344.791,-74.020,-176.158,7.774,148.379
C06988=1203.544,344.543,-73.989,-176.161,7.771,148.379
C06989=1203.548,344.295,-73.956,-176.162,7.768,148.379
C06990=1203.552,344.047,-73.923,-176.165,7.765,148.379
C06991=1203.557,343.800,-73.891,-176.167,7.762,148.378
C06992=1203.561,343.552,-73.859,-176.168,7.759,148.378
C06993=1203.564,343.304,-73.826,-176.171,7.756,148.378
C06994=1203.569,343.056,-73.794,-176.173,7.752,148.378
C06995=1203.573,342.808,-73.763,-176.175,7.750,148.378
C06996=1203.578,342.560,-73.730,-176.177,7.747,148.377
C06997=1203.581,342.313,-73.698,-176.179,7.743,148.377
C06998=1203.585,342.064,-73.665,-176.181,7.741,148.377
C06999=1203.590,341.817,-73.634,-176.183,7.738,148.377
C07000=1203.594,341.569,-73.601,-176.186,7.734,148.377
C07001=1203.598,341.321,-73.569,-176.187,7.732,148.376
C07002=1203.603,341.043,-73.533,-176.189,7.728,148.376
C07003=1203.607,340.764,-73.497,-176.192,7.725,148.376
C07004=1203.612,340.486,-73.460,-176.195,7.721,148.376
C07005=1203.617,340.208,-73.424,-176.197,7.718,148.376
C07006=1203.621,339.960,-73.392,-176.199,7.715,148.376
C07007=1203.626,339.712,-73.360,-176.201,7.712,148.375
C07008=1203.629,339.464,-73.328,-176.204,7.709,148.375
C07009=1203.633,339.216,-73.296,-176.205,7.706,148.375
C07010=1203.638,338.968,-73.264,-176.208,7.703,148.375
C07011=1203.642,338.720,-73.232,-176.210,7.700,148.375
C07012=1203.646,338.472,-73.200,-176.211,7.697,148.375
C07013=1203.650,338.224,-73.168,-176.214,7.694,148.375
C07014=1203.654,337.977,-73.136,-176.216,7.691,148.374
C07015=1203.659,337.728,-73.104,-176.218,7.688,148.374
C07016=1203.662,337.480,-73.072,-176.220,7.685,148.374
C07017=1203.667,337.233,-73.041,-176.223,7.682,148.374
C07018=1203.671,336.985,-73.008,-176.225,7.680,148.374
C07019=1203.675,336.736,-72.976,-176.227,7.676,148.374
C07020=1203.679,336.489,-72.945,-176.229,7.673,148.373
C07021=1203.684,336.241,-72.912,-176.231,7.671,148.373
C07022=1203.687,335.993,-72.881,-176.233,7.667,148.373
C07023=1203.692,335.745,-72.849,-176.236,7.664,148.373
C07024=1203.696,335.497,-72.817,-176.238,7.662,148.373
C07025=1203.700,335.250,-72.785,-176.240,7.658,148.373
C07026=1203.704,335.002,-72.753,-176.242,7.656,148.373
C07027=1203.709,334.753,-72.721,-176.244,7.653,148.373
C07028=1203.713,334.506,-72.689,-176.246,7.650,148.372
C07029=1203.717,334.257,-72.658,-176.248,7.647,148.372
C07030=1203.721,334.009,-72.627,-176.251,7.644,148.372
C07031=1203.726,333.762,-72.594,-176.253,7.641,148.372
C07032=1203.729,333.514,-72.563,-176.255,7.638,148.372
C07033=1203.734,333.266,-72.531,-176.257,7.635,148.372
C07034=1203.737,333.018,-72.499,-176.260,7.632,148.372
C07035=1203.742,332.769,-72.468,-176.261,7.629,148.371
C07036=1203.746,332.522,-72.436,-176.264,7.626,148.371
C07037=1203.750,332.274,-72.404,-176.266,7.623,148.371
C07038=1203.754,332.027,-72.373,-176.268,7.621,148.371
C07039=1203.758,331.778,-72.342,-176.270,7.617,148.371
C07040=1203.764,331.530,-72.310,-176.273,7.614,148.371
C07041=1203.767,331.282,-72.278,-176.275,7.612,148.371
C07042=1203.772,331.035,-72.246,-176.277,7.609,148.371
C07043=1203.776,330.786,-72.215,-176.280,7.605,148.371
C07044=1203.779,330.538,-72.183,-176.281,7.603,148.370
C07045=1203.784,330.291,-72.151,-176.284,7.600,148.370
C07046=1203.788,330.042,-72.120,-176.286,7.597,148.370
C07047=1203.793,329.795,-72.089,-176.288,7.594,148.370
C07048=1203.797,329.546,-72.057,-176.291,7.591,148.370
C07049=1203.801,329.299,-72.026,-176.293,7.588,148.370
C07050=1203.805,329.050,-71.994,-176.295,7.586,148.370
C07051=1203.809,328.803,-71.963,-176.297,7.582,148.370
C07052=1203.813,328.554,-71.931,-176.300,7.579,148.370
C07053=1203.818,328.307,-71.901,-176.302,7.577,148.369
C07054=1203.822,328.058,-71.868,-176.304,7.574,148.369
C07055=1203.826,327.811,-71.837,-176.306,7.570,148.369
C07056=1203.830,327.562,-71.806,-176.309,7.568,148.369
C07057=1203.835,327.315,-71.774,-176.311,7.565,148.369
C07058=1203.839,327.066,-71.743,-176.313,7.562,148.369
C07059=1203.843,326.819,-71.712,-176.315,7.559,148.369
C07060=1203.847,326.570,-71.680,-176.318,7.556,148.369
C07061=1203.851,326.323,-71.649,-176.320,7.553,148.369
C07062=1203.855,326.074,-71.618,-176.322,7.551,148.369
C07063=1203.860,325.826,-71.587,-176.324,7.547,148.369
C07064=1203.864,325.578,-71.555,-176.327,7.544,148.369
C07065=1203.868,325.330,-71.524,-176.329,7.542,148.369
C07066=1203.873,325.083,-71.493,-176.331,7.539,148.368
C07067=1203.877,324.834,-71.462,-176.334,7.536,148.368
C07068=1203.881,324.587,-71.430,-176.336,7.533,148.368
C07069=1203.885,324.338,-71.399,-176.338,7.530,148.368
C07070=1203.889,324.090,-71.368,-176.341,7.527,148.368
C07071=1203.893,323.842,-71.337,-176.343,7.525,148.368
C07072=1203.897,323.595,-71.306,-176.345,7.522,148.368
C07073=1203.902,323.347,-71.276,-176.348,7.518,148.368
C07074=1203.905,323.099,-71.244,-176.350,7.516,148.368
C07075=1203.910,322.851,-71.213,-176.352,7.513,148.368
C07076=1203.914,322.602,-71.182,-176.355,7.510,148.368
C07077=1203.919,322.354,-71.151,-176.357,7.507,148.368
C07078=1203.923,322.107,-71.120,-176.359,7.504,148.367
C07079=1203.927,321.858,-71.089,-176.361,7.502,148.368
C07080=1203.932,321.610,-71.058,-176.364,7.499,148.368
C07081=1203.936,321.361,-71.027,-176.366,7.496,148.367
C07082=1203.939,321.114,-70.996,-176.368,7.493,148.367
C07083=1203.944,320.866,-70.965,-176.370,7.490,148.367
C07084=1203.948,320.618,-70.934,-176.373,7.487,148.367
C07085=1203.952,320.370,-70.903,-176.375,7.485,148.367
C07086=1203.957,320.122,-70.872,-176.377,7.481,148.367
C07087=1203.961,319.874,-70.841,-176.380,7.478,148.367
C07088=1203.965,319.626,-70.810,-176.382,7.476,148.367
C07089=1203.969,319.378,-70.780,-176.384,7.473,148.367
C07090=1203.973,319.130,-70.748,-176.387,7.470,148.367
C07091=1203.978,318.882,-70.718,-176.389,7.468,148.367
C07092=1203.982,318.634,-70.688,-176.392,7.465,148.367
C07093=1203.986,318.385,-70.656,-176.394,7.461,148.367
C07094=1203.990,318.137,-70.626,-176.396,7.459,148.367
C07095=1203.995,317.889,-70.595,-176.399,7.456,148.367
C07096=1203.999,317.641,-70.564,-176.401,7.453,148.367
C07097=1204.003,317.393,-70.534,-176.403,7.451,148.367
C07098=1204.007,317.145,-70.503,-176.406,7.447,148.367
C07099=1204.011,316.896,-70.472,-176.408,7.445,148.367
C07100=1204.015,316.649,-70.442,-176.410,7.442,148.366
C07101=1204.020,316.401,-70.411,-176.413,7.439,148.366
C07102=1204.025,316.153,-70.380,-176.415,7.437,148.366
C07103=1204.029,315.904,-70.349,-176.417,7.433,148.366
C07104=1204.032,315.657,-70.319,-176.420,7.430,148.366
C07105=1204.037,315.409,-70.288,-176.422,7.428,148.366
C07106=1204.042,315.133,-70.254,-176.425,7.425,148.366
C07107=1204.046,314.856,-70.220,-176.428,7.422,148.366
C07108=1204.051,314.580,-70.185,-176.431,7.418,148.366
C07109=1204.056,314.304,-70.151,-176.433,7.415,148.366
C07110=1204.060,314.056,-70.122,-176.435,7.413,148.366
C07111=1204.064,313.807,-70.091,-176.438,7.410,148.366
C07112=1204.069,313.559,-70.060,-176.440,7.407,148.366
C07113=1204.073,313.312,-70.030,-176.443,7.404,148.366
C07114=1204.077,313.064,-69.999,-176.445,7.401,148.366
C07115=1204.081,312.816,-69.969,-176.447,7.399,148.366
C07116=1204.085,312.567,-69.938,-176.450,7.396,148.366
C07117=1204.090,312.319,-69.908,-176.452,7.393,148.366
C07118=1204.094,312.071,-69.877,-176.455,7.391,148.366
C07119=1204.098,311.823,-69.847,-176.457,7.387,148.366
C07120=1204.103,311.575,-69.817,-176.459,7.384,148.366
C07121=1204.107,311.326,-69.786,-176.462,7.382,148.366
C07122=1204.111,311.079,-69.756,-176.464,7.379,148.366
C07123=1204.115,310.831,-69.725,-176.466,7.377,148.366
C07124=1204.119,310.582,-69.696,-176.469,7.374,148.366
C07125=1204.124,310.334,-69.665,-176.471,7.371,148.366
C07126=1204.128,310.087,-69.635,-176.473,7.368,148.366
C07127=1204.132,309.837,-69.604,-176.476,7.365,148.366
C07128=1204.136,309.590,-69.574,-176.479,7.362,148.366
C07129=1204.141,309.342,-69.543,-176.481,7.360,148.366
C07130=1204.145,309.094,-69.514,-176.484,7.357,148.366
C07131=1204.149,308.846,-69.483,-176.486,7.355,148.366
C07132=1204.154,308.597,-69.454,-176.488,7.352,148.366
C07133=1204.158,308.349,-69.423,-176.491,7.348,148.366
C07134=1204.161,308.101,-69.392,-176.493,7.346,148.366
C07135=1204.166,307.852,-69.362,-176.495,7.343,148.366
C07136=1204.170,307.605,-69.332,-176.498,7.341,148.366
C07137=1204.175,307.356,-69.302,-176.500,7.338,148.366
C07138=1204.179,307.109,-69.272,-176.503,7.335,148.366
C07139=1204.183,306.860,-69.243,-176.505,7.333,148.366
C07140=1204.188,306.612,-69.212,-176.508,7.330,148.366
C07141=1204.192,306.364,-69.182,-176.510,7.326,148.366
C07142=1204.197,306.116,-69.152,-176.512,7.324,148.366
C07143=1204.201,305.868,-69.122,-176.515,7.321,148.366
C07144=1204.205,305.620,-69.092,-176.517,7.319,148.366
C07145=1204.210,305.372,-69.062,-176.520,7.316,148.366
C07146=1204.213,305.123,-69.032,-176.522,7.313,148.366
C07147=1204.217,304.875,-69.002,-176.524,7.311,148.366
C07148=1204.222,304.626,-68.972,-176.527,7.308,148.366
C07149=1204.226,304.379,-68.942,-176.529,7.306,148.366
C07150=1204.230,304.131,-68.912,-176.532,7.303,148.366
C07151=1204.235,303.882,-68.882,-176.535,7.300,148.366
C07152=1204.239,303.634,-68.852,-176.537,7.297,148.366
C07153=1204.243,303.386,-68.823,-176.539,7.294,148.366
C07154=1204.248,303.137,-68.792,-176.542,7.292,148.366
C07155=1204.252,302.890,-68.762,-176.544,7.289,148.366
C07156=1204.256,302.642,-68.733,-176.547,7.286,148.366
C07157=1204.261,302.393,-68.703,-176.549,7.284,148.366
C07158=1204.265,302.145,-68.673,-176.552,7.281,148.366
C07159=1204.269,301.897,-68.643,-176.554,7.279,148.366
C07160=1204.273,301.649,-68.614,-176.557,7.276,148.366
C07161=1204.278,301.400,-68.584,-176.559,7.273,148.366
C07162=1204.282,301.152,-68.554,-176.561,7.270,148.367
C07163=1204.286,300.904,-68.524,-176.564,7.267,148.367
C07164=1204.290,300.656,-68.495,-176.566,7.265,148.367
C07165=1204.295,300.408,-68.465,-176.569,7.262,148.367
C07166=1204.299,300.159,-68.435,-176.572,7.259,148.367
C07167=1204.304,299.911,-68.406,-176.574,7.257,148.367
C07168=1204.308,299.663,-68.376,-176.576,7.254,148.367
C07169=1204.312,299.415,-68.346,-176.579,7.252,148.367
C07170=1204.316,299.167,-68.317,-176.581,7.249,148.367
C07171=1204.321,298.919,-68.288,-176.583,7.247,148.367
C07172=1204.326,298.671,-68.257,-176.586,7.244,148.367
C07173=1204.330,298.422,-68.228,-176.589,7.240,148.367
C07174=1204.334,298.174,-68.199,-176.591,7.238,148.367
C07175=1204.338,297.926,-68.169,-176.594,7.235,148.367
C07176=1204.342,297.678,-68.140,-176.596,7.233,148.367
C07177=1204.346,297.429,-68.110,-176.598,7.230,148.367
C07178=1204.351,297.181,-68.081,-176.601,7.228,148.367
C07179=1204.355,296.933,-68.051,-176.603,7.225,148.367
C07180=1204.359,296.684,-68.022,-176.606,7.222,148.367
C07181=1204.364,296.436,-67.992,-176.608,7.220,148.367
C07182=1204.368,296.188,-67.962,-176.611,7.217,148.367
C07183=1204.373,295.940,-67.933,-176.613,7.214,148.367
C07184=1204.377,295.692,-67.904,-176.616,7.211,148.367
C07185=1204.381,295.444,-67.874,-176.618,7.209,148.367
C07186=1204.385,295.195,-67.845,-176.620,7.206,148.367
C07187=1204.390,294.947,-67.815,-176.623,7.203,148.367
C07188=1204.394,294.699,-67.786,-176.626,7.201,148.368
C07189=1204.398,294.450,-67.757,-176.628,7.198,148.368
C07190=1204.402,294.202,-67.727,-176.631,7.196,148.368
C07191=1204.407,293.955,-67.698,-176.633,7.193,148.368
C07192=1204.411,293.706,-67.669,-176.635,7.191,148.368
C07193=1204.416,293.457,-67.640,-176.638,7.188,148.368
C07194=1204.420,293.209,-67.610,-176.640,7.186,148.368
C07195=1204.424,292.961,-67.581,-176.643,7.183,148.368
C07196=1204.428,292.713,-67.551,-176.646,7.180,148.368
C07197=1204.433,292.465,-67.522,-176.648,7.177,148.368
C07198=1204.437,292.217,-67.494,-176.651,7.175,148.368
C07199=1204.441,291.968,-67.465,-176.653,7.172,148.368
C07200=1204.445,291.720,-67.435,-176.656,7.169,148.368
C07201=1204.449,291.472,-67.406,-176.658,7.167,148.368
C07202=1204.454,291.224,-67.377,-176.661,7.164,148.369
C07203=1204.459,290.975,-67.348,-176.663,7.162,148.369
C07204=1204.463,290.727,-67.319,-176.665,7.159,148.369
C07205=1204.467,290.479,-67.289,-176.667,7.157,148.369
C07206=1204.471,290.230,-67.260,-176.671,7.154,148.369
C07207=1204.476,289.982,-67.231,-176.673,7.152,148.369
C07208=1204.480,289.734,-67.202,-176.675,7.149,148.369
C07209=1204.484,289.485,-67.174,-176.678,7.146,148.369
C07210=1204.489,289.211,-67.141,-176.680,7.144,148.369
C07211=1204.494,288.937,-67.109,-176.683,7.141,148.369
C07212=1204.499,288.663,-67.077,-176.686,7.138,148.369
C07213=1204.504,288.388,-67.046,-176.689,7.135,148.369
C07214=1204.508,288.140,-67.016,-176.692,7.132,148.369
C07215=1204.512,287.892,-66.987,-176.694,7.130,148.369
C07216=1204.516,287.643,-66.959,-176.697,7.127,148.370
C07217=1204.521,287.396,-66.930,-176.699,7.125,148.370
C07218=1204.525,287.147,-66.901,-176.702,7.122,148.370
C07219=1204.529,286.898,-66.871,-176.704,7.120,148.370
C07220=1204.534,286.650,-66.843,-176.706,7.117,148.370
C07221=1204.538,286.402,-66.814,-176.709,7.115,148.370
C07222=1204.542,286.153,-66.786,-176.712,7.112,148.370
C07223=1204.546,285.905,-66.756,-176.714,7.110,148.370
C07224=1204.552,285.657,-66.728,-176.717,7.107,148.370
C07225=1204.555,285.409,-66.699,-176.719,7.104,148.370
C07226=1204.560,285.160,-66.670,-176.722,7.102,148.371
C07227=1204.565,284.912,-66.642,-176.724,7.099,148.371
C07228=1204.568,284.664,-66.613,-176.727,7.096,148.371
C07229=1204.573,284.415,-66.584,-176.729,7.094,148.371
C07230=1204.577,284.168,-66.555,-176.732,7.091,148.371
C07231=1204.582,283.919,-66.526,-176.734,7.089,148.371
C07232=1204.586,283.670,-66.498,-176.737,7.086,148.371
C07233=1204.590,283.423,-66.469,-176.739,7.084,148.371
C07234=1204.594,283.174,-66.441,-176.742,7.081,148.371
C07235=1204.599,282.925,-66.412,-176.744,7.079,148.371
C07236=1204.603,282.677,-66.383,-176.747,7.076,148.372
C07237=1204.607,282.429,-66.355,-176.749,7.074,148.372
C07238=1204.612,282.181,-66.327,-176.752,7.071,148.372
C07239=1204.616,281.932,-66.297,-176.754,7.069,148.372
C07240=1204.620,281.684,-66.269,-176.757,7.066,148.372
C07241=1204.625,281.436,-66.241,-176.759,7.064,148.372
C07242=1204.629,281.187,-66.212,-176.762,7.061,148.372
C07243=1204.634,280.940,-66.183,-176.764,7.059,148.372
C07244=1204.638,280.691,-66.155,-176.767,7.056,148.372
C07245=1204.642,280.442,-66.127,-176.769,7.054,148.372
C07246=1204.647,280.194,-66.098,-176.772,7.051,148.372
C07247=1204.651,279.945,-66.070,-176.774,7.049,148.373
C07248=1204.656,279.698,-66.041,-176.777,7.046,148.373
C07249=1204.659,279.449,-66.013,-176.780,7.044,148.373
C07250=1204.664,279.200,-65.984,-176.782,7.042,148.373
C07251=1204.668,278.952,-65.956,-176.784,7.039,148.373
C07252=1204.673,278.704,-65.928,-176.787,7.037,148.373
C07253=1204.677,278.456,-65.900,-176.790,7.034,148.373
C07254=1204.682,278.207,-65.871,-176.792,7.032,148.373
C07255=1204.686,277.959,-65.843,-176.795,7.029,148.374
C07256=1204.690,277.711,-65.814,-176.797,7.027,148.374
C07257=1204.694,277.463,-65.786,-176.800,7.024,148.374
C07258=1204.699,277.214,-65.757,-176.802,7.021,148.374
C07259=1204.703,276.966,-65.729,-176.805,7.019,148.374
C07260=1204.708,276.717,-65.701,-176.807,7.017,148.374
C07261=1204.712,276.469,-65.673,-176.810,7.014,148.374
C07262=1204.716,276.221,-65.645,-176.813,7.012,148.374
C07263=1204.721,275.972,-65.616,-176.815,7.009,148.375
C07264=1204.725,275.724,-65.588,-176.817,7.006,148.375
C07265=1204.730,275.476,-65.560,-176.820,7.005,148.375
C07266=1204.733,275.227,-65.532,-176.823,7.002,148.375
C07267=1204.738,274.979,-65.504,-176.825,6.999,148.375
C07268=1204.743,274.730,-65.476,-176.828,6.996,148.375
C07269=1204.747,274.482,-65.448,-176.830,6.995,148.375
C07270=1204.751,274.233,-65.419,-176.833,6.991,148.375
C07271=1204.756,273.985,-65.392,-176.835,6.989,148.375
C07272=1204.760,273.737,-65.364,-176.838,6.987,148.376
C07273=1204.765,273.488,-65.335,-176.840,6.984,148.376
C07274=1204.768,273.240,-65.307,-176.843,6.982,148.376
C07275=1204.773,272.992,-65.279,-176.846,6.980,148.376
C07276=1204.778,272.742,-65.251,-176.848,6.977,148.376
C07277=1204.782,272.494,-65.223,-176.851,6.974,148.376
C07278=1204.786,272.247,-65.196,-176.853,6.972,148.377
C07279=1204.791,271.998,-65.167,-176.855,6.970,148.377
C07280=1204.795,271.750,-65.139,-176.858,6.967,148.377
C07281=1204.799,271.501,-65.112,-176.861,6.965,148.377
C07282=1204.804,271.253,-65.084,-176.863,6.962,148.377
C07283=1204.808,271.004,-65.055,-176.866,6.961,148.377
C07284=1204.812,270.756,-65.027,-176.868,6.958,148.377
C07285=1204.817,270.508,-65.000,-176.871,6.955,148.377
C07286=1204.821,270.259,-64.972,-176.873,6.953,148.378
C07287=1204.826,270.011,-64.944,-176.876,6.950,148.378
C07288=1204.830,269.762,-64.916,-176.878,6.948,148.378
C07289=1204.834,269.514,-64.889,-176.881,6.946,148.378
C07290=1204.839,269.266,-64.861,-176.884,6.943,148.378
C07291=1204.843,269.017,-64.832,-176.886,6.941,148.378
C07292=1204.848,268.768,-64.805,-176.889,6.939,148.378
C07293=1204.852,268.521,-64.777,-176.891,6.936,148.379
C07294=1204.856,268.271,-64.750,-176.894,6.934,148.379
C07295=1204.861,268.023,-64.722,-176.896,6.931,148.379
C07296=1204.865,267.776,-64.694,-176.898,6.929,148.379
C07297=1204.870,267.526,-64.666,-176.902,6.927,148.379
C07298=1204.874,267.278,-64.639,-176.904,6.924,148.379
C07299=1204.879,267.030,-64.611,-176.906,6.923,148.380
C07300=1204.882,266.781,-64.583,-176.909,6.920,148.380
C07301=1204.887,266.533,-64.556,-176.911,6.917,148.380
C07302=1204.891,266.285,-64.528,-176.914,6.915,148.380
C07303=1204.895,266.036,-64.501,-176.917,6.912,148.380
C07304=1204.901,265.787,-64.473,-176.919,6.911,148.380
